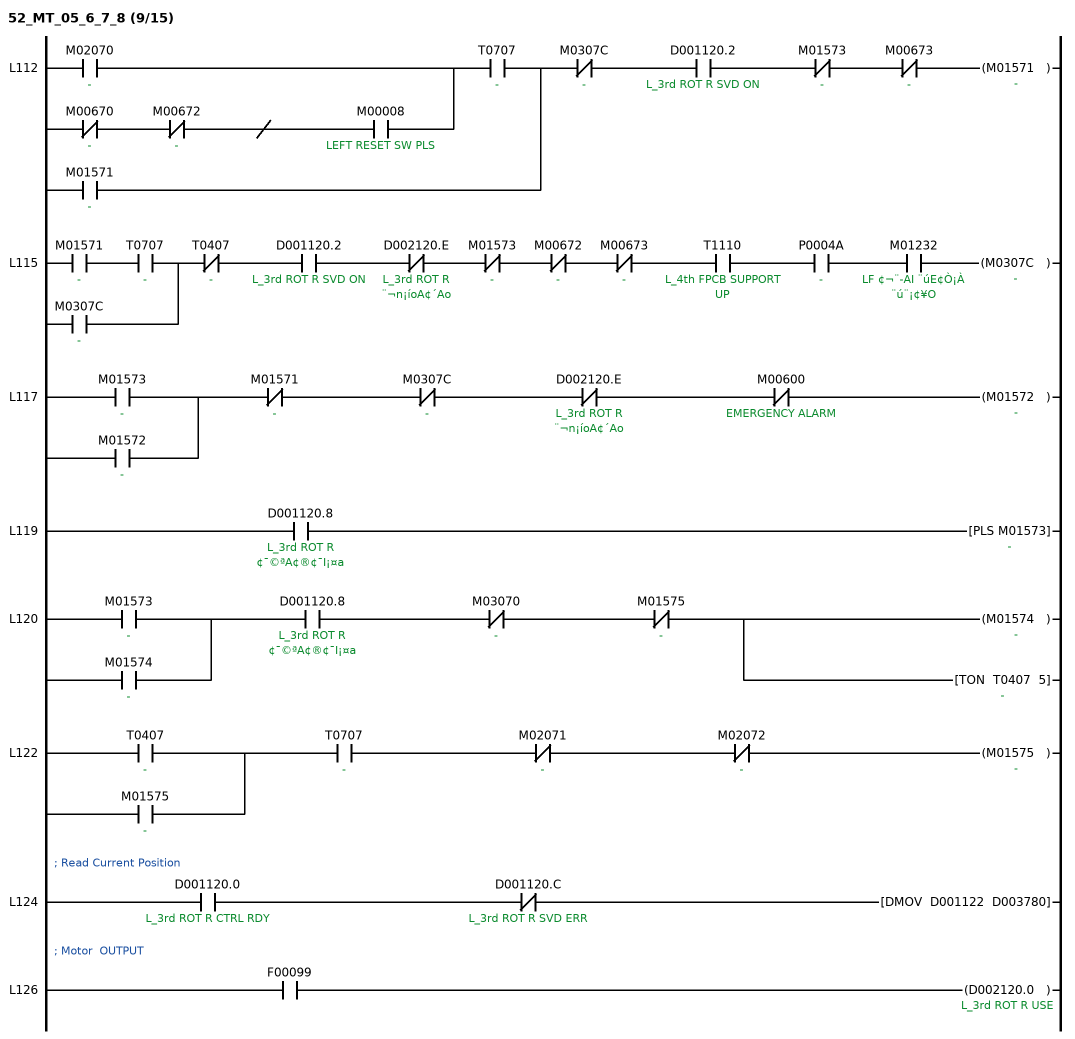
[picture p264: 52_MT_05_6_7_8 rungs L112-L126]
; L112
LOAD      M02070	// -
LOAD NOT  M00670	// -
AND NOT   M00672	// -
NOT
AND       M00008	// LEFT RESET SW PLS
OR LOAD
AND       T0707	// -
OR        M01571	// -
AND NOT   M0307C	// -
AND       D001120.2	// L_3rd ROT R SVD ON
AND NOT   M01573	// -
AND NOT   M00673	// -
OUT       M01571	// -
; L115
LOAD      M01571	// -
AND       T0707	// -
OR        M0307C	// -
AND NOT   T0407	// -
AND       D001120.2	// L_3rd ROT R SVD ON
AND NOT   D002120.E	// L_3rd ROT R ¨¬n¡íoA¢´Ao
AND NOT   M01573	// -
AND NOT   M00672	// -
AND NOT   M00673	// -
AND       T1110	// L_4th FPCB SUPPORT UP
AND       P0004A	// -
AND       M01232	// LF ¢¬¨­AI ¨úE¢Ò¡À ¨ú¨¡¢¥O
OUT       M0307C	// -
; L117
LOAD      M01573	// -
OR        M01572	// -
AND NOT   M01571	// -
AND NOT   M0307C	// -
AND NOT   D002120.E	// L_3rd ROT R ¨¬n¡íoA¢´Ao
AND NOT   M00600	// EMERGENCY ALARM
OUT       M01572	// -
; L119
LOAD      D001120.8	// L_3rd ROT R ¢¯©ªA¢®¢¯I¡¤a
OUTP      M01573	// -
; L120
LOAD      M01573	// -
OR        M01574	// -
AND       D001120.8	// L_3rd ROT R ¢¯©ªA¢®¢¯I¡¤a
AND NOT   M03070	// -
AND NOT   M01575	// -
OUT       M01574	// -
TON       T0407 5	// -
; L122
LOAD      T0407	// -
OR        M01575	// -
AND       T0707	// -
AND NOT   M02071	// -
AND NOT   M02072	// -
OUT       M01575	// -
; L124
LOAD      D001120.0	// L_3rd ROT R CTRL RDY
AND NOT   D001120.C	// L_3rd ROT R SVD ERR
DMOV      D001122 D003780
// output comment: Read Current Position
//  Motor  OUTPUT
; L126
LOAD      F00099
OUT       D002120.0	// L_3rd ROT R USE

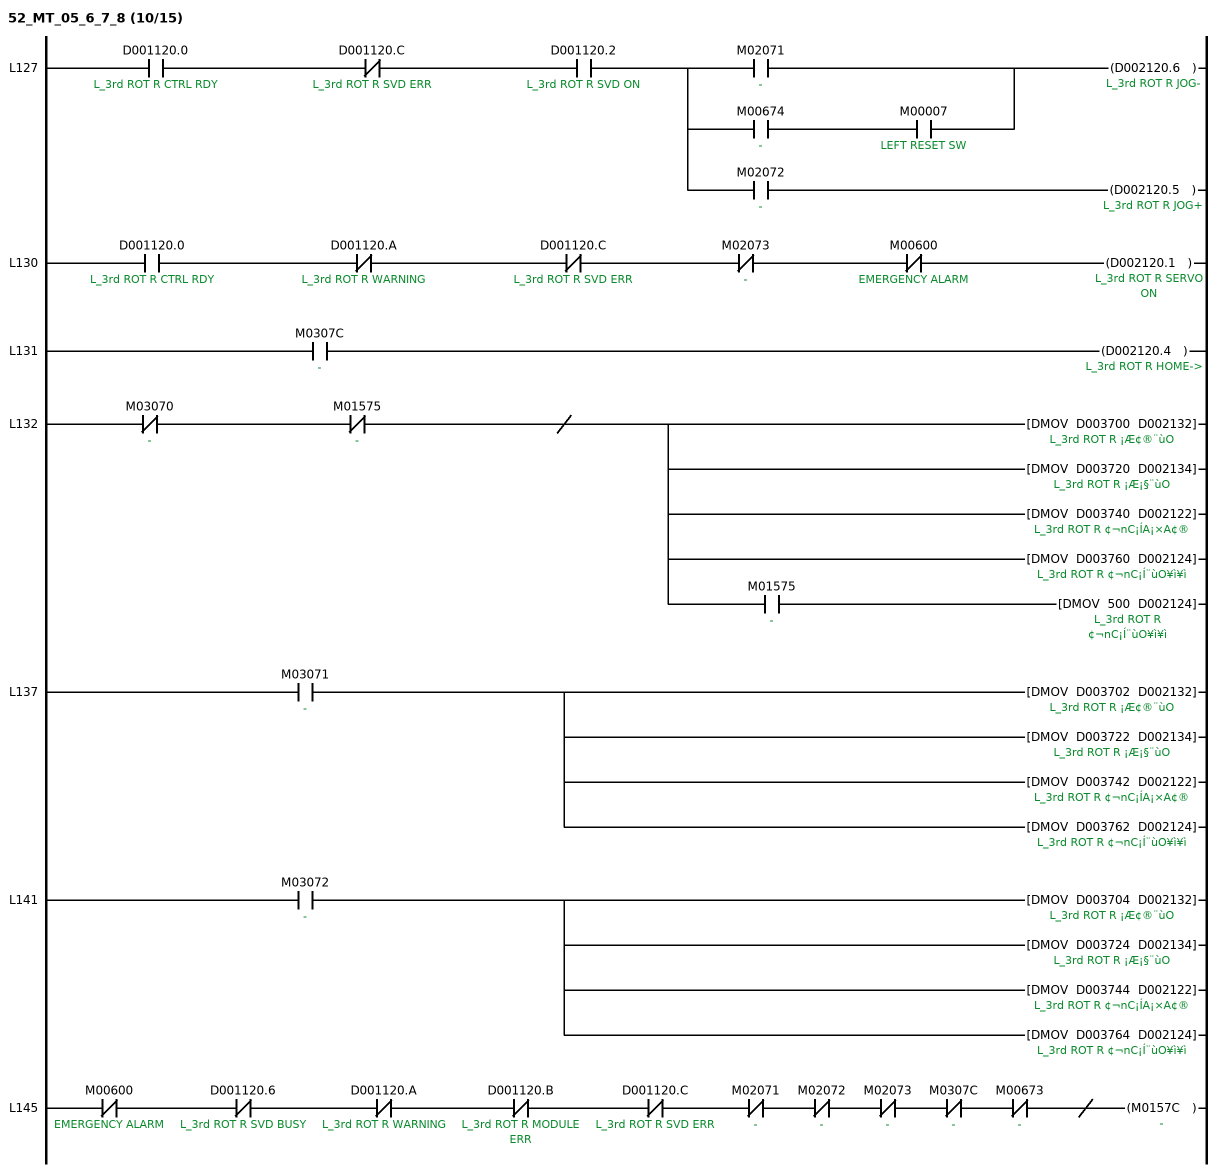
; L127
LOAD      D001120.0	// L_3rd ROT R CTRL RDY
AND NOT   D001120.C	// L_3rd ROT R SVD ERR
AND       D001120.2	// L_3rd ROT R SVD ON
MPUSH
LOAD      M02071	// -
LOAD      M00674	// -
AND       M00007	// LEFT RESET SW
OR LOAD
AND LOAD
OUT       D002120.6	// L_3rd ROT R JOG-
MPOP
AND       M02072	// -
OUT       D002120.5	// L_3rd ROT R JOG+
; L130
LOAD      D001120.0	// L_3rd ROT R CTRL RDY
AND NOT   D001120.A	// L_3rd ROT R WARNING
AND NOT   D001120.C	// L_3rd ROT R SVD ERR
AND NOT   M02073	// -
AND NOT   M00600	// EMERGENCY ALARM
OUT       D002120.1	// L_3rd ROT R SERVO ON
; L131
LOAD      M0307C	// -
OUT       D002120.4	// L_3rd ROT R HOME->
; L132
LOAD NOT  M03070	// -
AND NOT   M01575	// -
NOT
DMOV      D003700 D002132	// L_3rd ROT R ¡Æ¢®¨ùO
DMOV      D003720 D002134	// L_3rd ROT R ¡Æ¡§¨ùO
DMOV      D003740 D002122	// L_3rd ROT R ¢¬nC¡ÍA¡×A¢®
DMOV      D003760 D002124	// L_3rd ROT R ¢¬nC¡Í¨ùO¥ì¥ì
AND       M01575	// -
DMOV      500 D002124	// L_3rd ROT R ¢¬nC¡Í¨ùO¥ì¥ì
; L137
LOAD      M03071	// -
DMOV      D003702 D002132	// L_3rd ROT R ¡Æ¢®¨ùO
DMOV      D003722 D002134	// L_3rd ROT R ¡Æ¡§¨ùO
DMOV      D003742 D002122	// L_3rd ROT R ¢¬nC¡ÍA¡×A¢®
DMOV      D003762 D002124	// L_3rd ROT R ¢¬nC¡Í¨ùO¥ì¥ì
; L141
LOAD      M03072	// -
DMOV      D003704 D002132	// L_3rd ROT R ¡Æ¢®¨ùO
DMOV      D003724 D002134	// L_3rd ROT R ¡Æ¡§¨ùO
DMOV      D003744 D002122	// L_3rd ROT R ¢¬nC¡ÍA¡×A¢®
DMOV      D003764 D002124	// L_3rd ROT R ¢¬nC¡Í¨ùO¥ì¥ì
; L145
LOAD NOT  M00600	// EMERGENCY ALARM
AND NOT   D001120.6	// L_3rd ROT R SVD BUSY
AND NOT   D001120.A	// L_3rd ROT R WARNING
AND NOT   D001120.B	// L_3rd ROT R MODULE ERR
AND NOT   D001120.C	// L_3rd ROT R SVD ERR
AND NOT   M02071	// -
AND NOT   M02072	// -
AND NOT   M02073	// -
AND NOT   M0307C	// -
AND NOT   M00673	// -
NOT
OUT       M0157C	// -

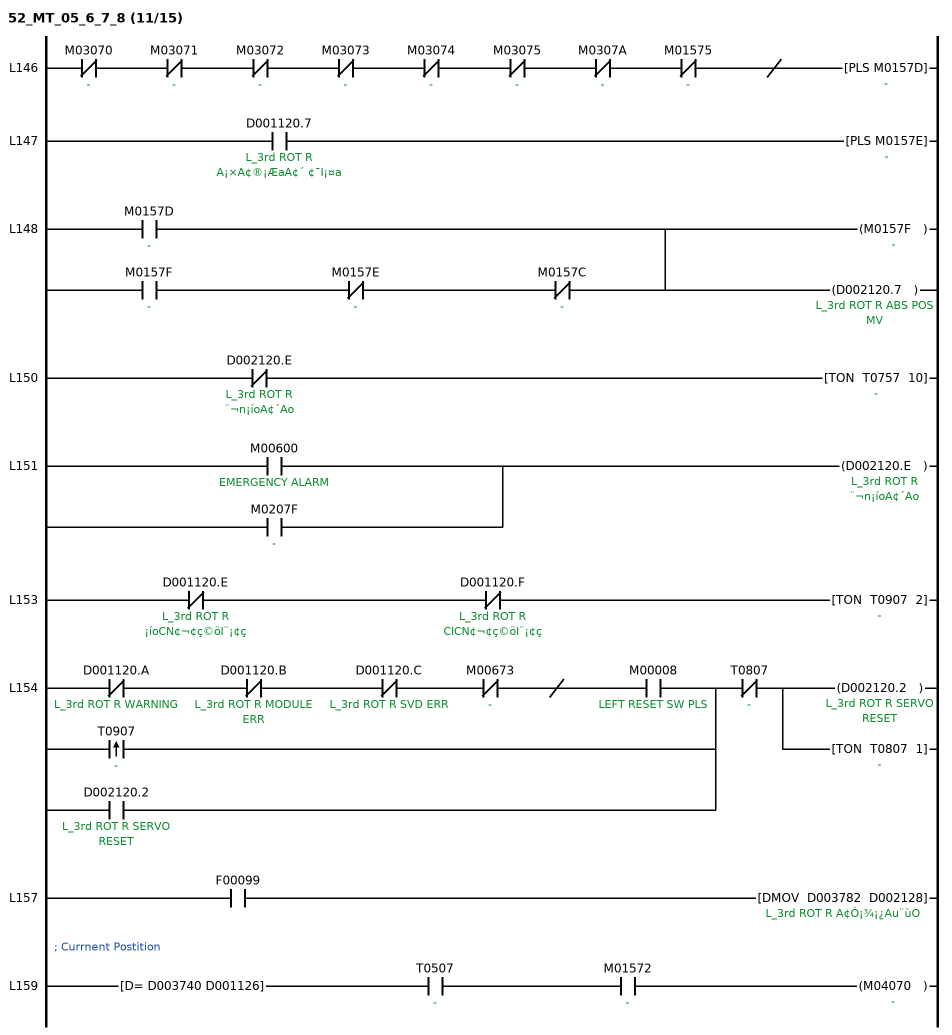
; L146
LOAD NOT  M03070	// -
AND NOT   M03071	// -
AND NOT   M03072	// -
AND NOT   M03073	// -
AND NOT   M03074	// -
AND NOT   M03075	// -
AND NOT   M0307A	// -
AND NOT   M01575	// -
NOT
OUTP      M0157D	// -
; L147
LOAD      D001120.7	// L_3rd ROT R A¡×A¢®¡ÆaA¢´ ¢¯I¡¤a
OUTP      M0157E	// -
; L148
LOAD      M0157D	// -
LOAD      M0157F	// -
AND NOT   M0157E	// -
AND NOT   M0157C	// -
OR LOAD
OUT       M0157F	// -
OUT       D002120.7	// L_3rd ROT R ABS POS MV
; L150
LOAD NOT  D002120.E	// L_3rd ROT R ¨¬n¡íoA¢´Ao
TON       T0757 10	// -
; L151
LOAD      M00600	// EMERGENCY ALARM
OR        M0207F	// -
OUT       D002120.E	// L_3rd ROT R ¨¬n¡íoA¢´Ao
; L153
LOAD NOT  D001120.E	// L_3rd ROT R ¡íoCN¢¬¢ç©öI¨¡¢ç
AND NOT   D001120.F	// L_3rd ROT R CICN¢¬¢ç©öI¨¡¢ç
TON       T0907 2	// -
; L154
LOAD NOT  D001120.A	// L_3rd ROT R WARNING
AND NOT   D001120.B	// L_3rd ROT R MODULE ERR
AND NOT   D001120.C	// L_3rd ROT R SVD ERR
AND NOT   M00673	// -
NOT
AND       M00008	// LEFT RESET SW PLS
ORP       T0907	// -
OR        D002120.2	// L_3rd ROT R SERVO RESET
AND NOT   T0807	// -
OUT       D002120.2	// L_3rd ROT R SERVO RESET
TON       T0807 1	// -
; L157
LOAD      F00099
DMOV      D003782 D002128	// L_3rd ROT R A¢Ò¡¾¡¿Au¨ùO
// Currnent Postition
; L159
LOADD=    D003740 D001126
AND       T0507	// -
AND       M01572	// -
OUT       M04070	// -

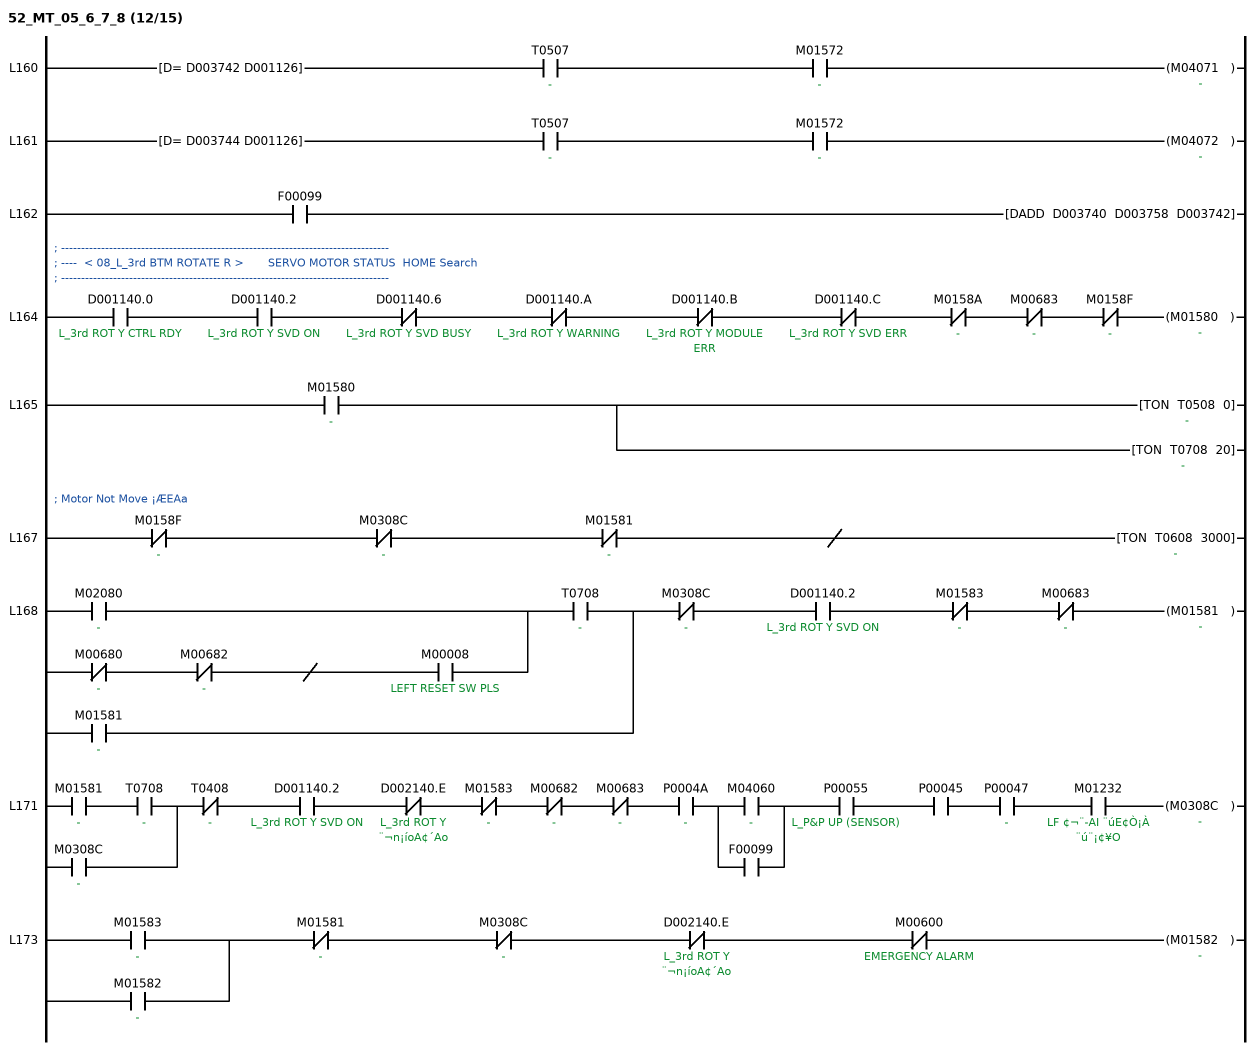
; L160
LOADD=    D003742 D001126
AND       T0507	// -
AND       M01572	// -
OUT       M04071	// -
; L161
LOADD=    D003744 D001126
AND       T0507	// -
AND       M01572	// -
OUT       M04072	// -
; L162
LOAD      F00099
DADD      D003740 D003758 D003742
// ----------------------------------------------------------------------------------
// 
// ----  < 08_L_3rd BTM ROTATE R >       SERVO MOTOR STATUS  HOME Search
// 
// ----------------------------------------------------------------------------------
; L164
LOAD      D001140.0	// L_3rd ROT Y CTRL RDY
AND       D001140.2	// L_3rd ROT Y SVD ON
AND NOT   D001140.6	// L_3rd ROT Y SVD BUSY
AND NOT   D001140.A	// L_3rd ROT Y WARNING
AND NOT   D001140.B	// L_3rd ROT Y MODULE ERR
AND NOT   D001140.C	// L_3rd ROT Y SVD ERR
AND NOT   M0158A	// -
AND NOT   M00683	// -
AND NOT   M0158F	// -
OUT       M01580	// -
; L165
LOAD      M01580	// -
TON       T0508 0	// -
TON       T0708 20	// -
; L167
LOAD NOT  M0158F	// -
AND NOT   M0308C	// -
AND NOT   M01581	// -
NOT
TON       T0608 3000	// -
// output comment: Motor Not Move ¡ÆEAa
; L168
LOAD      M02080	// -
LOAD NOT  M00680	// -
AND NOT   M00682	// -
NOT
AND       M00008	// LEFT RESET SW PLS
OR LOAD
AND       T0708	// -
OR        M01581	// -
AND NOT   M0308C	// -
AND       D001140.2	// L_3rd ROT Y SVD ON
AND NOT   M01583	// -
AND NOT   M00683	// -
OUT       M01581	// -
; L171
LOAD      M01581	// -
AND       T0708	// -
OR        M0308C	// -
AND NOT   T0408	// -
AND       D001140.2	// L_3rd ROT Y SVD ON
AND NOT   D002140.E	// L_3rd ROT Y ¨¬n¡íoA¢´Ao
AND NOT   M01583	// -
AND NOT   M00682	// -
AND NOT   M00683	// -
AND       P0004A	// -
LOAD      M04060	// -
OR        F00099
AND LOAD
AND       P00055	// L_P&P UP (SENSOR)
AND       P00045
AND       P00047	// -
AND       M01232	// LF ¢¬¨­AI ¨úE¢Ò¡À ¨ú¨¡¢¥O
OUT       M0308C	// -
; L173
LOAD      M01583	// -
OR        M01582	// -
AND NOT   M01581	// -
AND NOT   M0308C	// -
AND NOT   D002140.E	// L_3rd ROT Y ¨¬n¡íoA¢´Ao
AND NOT   M00600	// EMERGENCY ALARM
OUT       M01582	// -

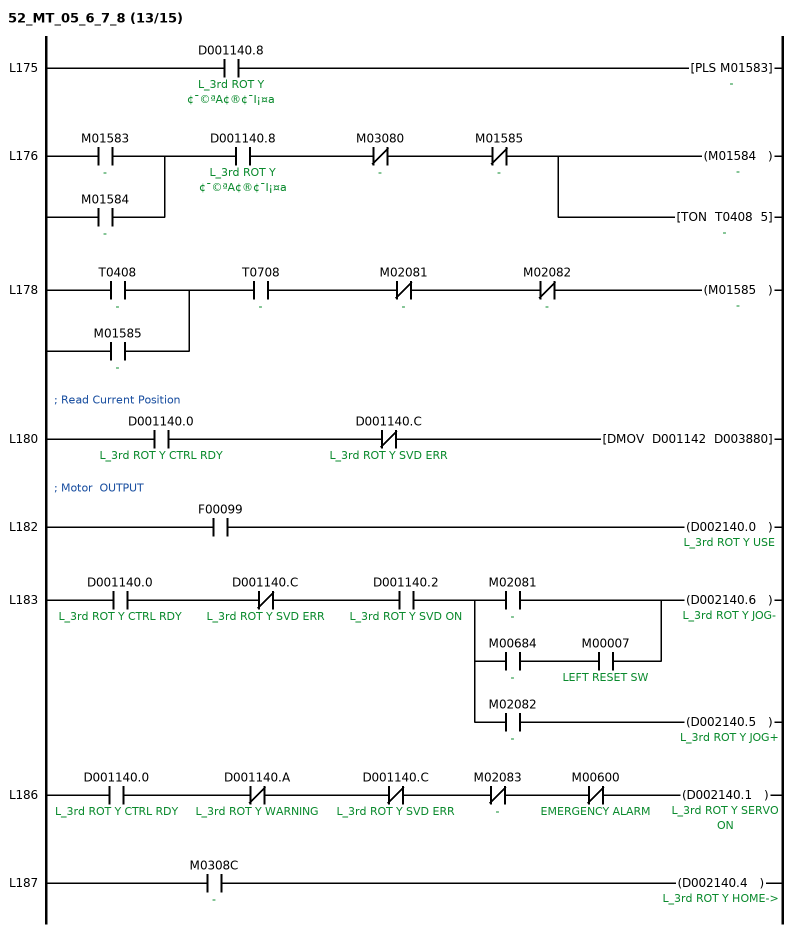
; L175
LOAD      D001140.8	// L_3rd ROT Y ¢¯©ªA¢®¢¯I¡¤a
OUTP      M01583	// -
; L176
LOAD      M01583	// -
OR        M01584	// -
AND       D001140.8	// L_3rd ROT Y ¢¯©ªA¢®¢¯I¡¤a
AND NOT   M03080	// -
AND NOT   M01585	// -
OUT       M01584	// -
TON       T0408 5	// -
; L178
LOAD      T0408	// -
OR        M01585	// -
AND       T0708	// -
AND NOT   M02081	// -
AND NOT   M02082	// -
OUT       M01585	// -
; L180
LOAD      D001140.0	// L_3rd ROT Y CTRL RDY
AND NOT   D001140.C	// L_3rd ROT Y SVD ERR
DMOV      D001142 D003880
// output comment: Read Current Position
//  Motor  OUTPUT
; L182
LOAD      F00099
OUT       D002140.0	// L_3rd ROT Y USE
; L183
LOAD      D001140.0	// L_3rd ROT Y CTRL RDY
AND NOT   D001140.C	// L_3rd ROT Y SVD ERR
AND       D001140.2	// L_3rd ROT Y SVD ON
MPUSH
LOAD      M02081	// -
LOAD      M00684	// -
AND       M00007	// LEFT RESET SW
OR LOAD
AND LOAD
OUT       D002140.6	// L_3rd ROT Y JOG-
MPOP
AND       M02082	// -
OUT       D002140.5	// L_3rd ROT Y JOG+
; L186
LOAD      D001140.0	// L_3rd ROT Y CTRL RDY
AND NOT   D001140.A	// L_3rd ROT Y WARNING
AND NOT   D001140.C	// L_3rd ROT Y SVD ERR
AND NOT   M02083	// -
AND NOT   M00600	// EMERGENCY ALARM
OUT       D002140.1	// L_3rd ROT Y SERVO ON
; L187
LOAD      M0308C	// -
OUT       D002140.4	// L_3rd ROT Y HOME->

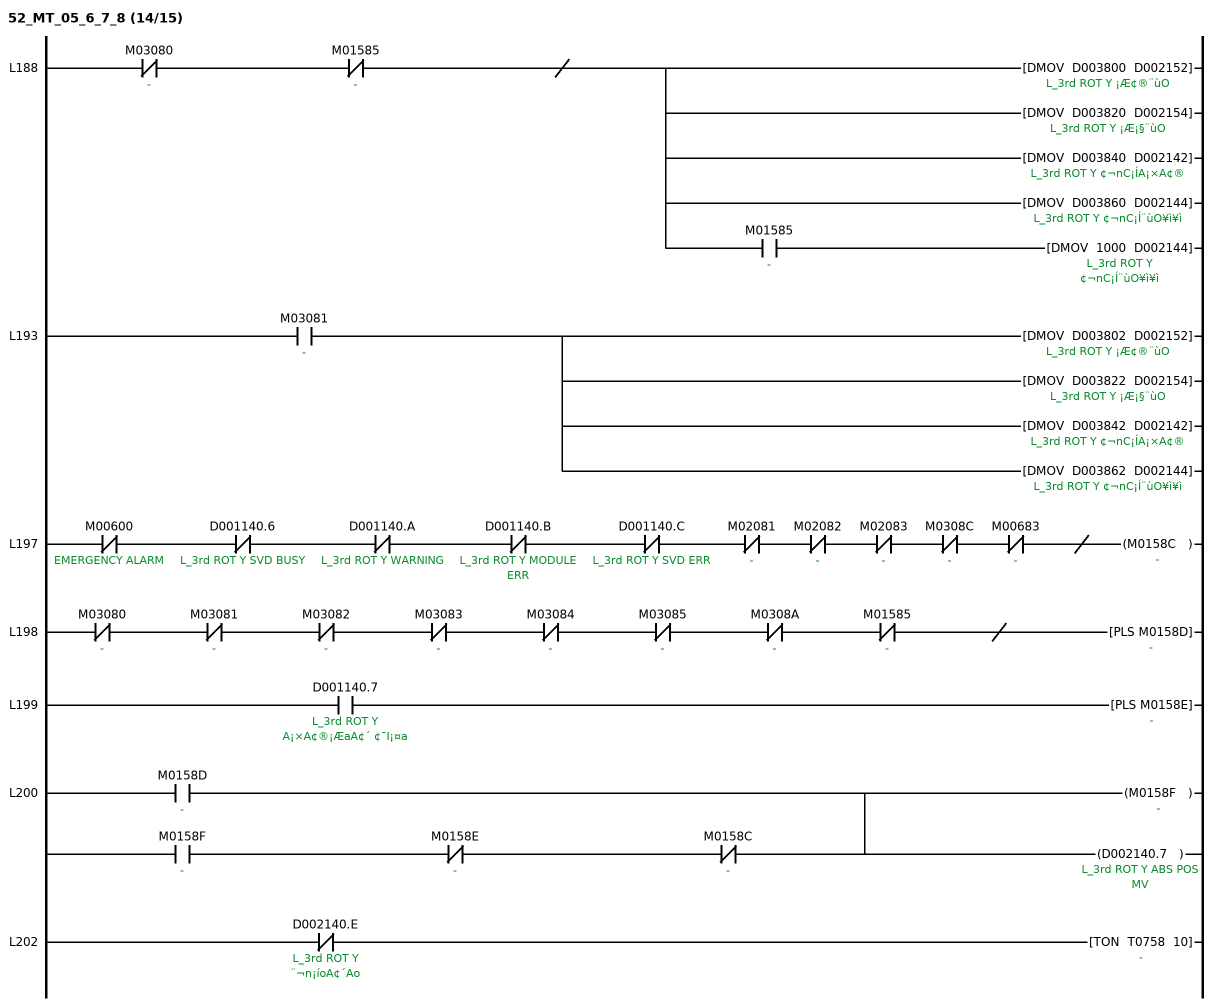
; L188
LOAD NOT  M03080	// -
AND NOT   M01585	// -
NOT
DMOV      D003800 D002152	// L_3rd ROT Y ¡Æ¢®¨ùO
DMOV      D003820 D002154	// L_3rd ROT Y ¡Æ¡§¨ùO
DMOV      D003840 D002142	// L_3rd ROT Y ¢¬nC¡ÍA¡×A¢®
DMOV      D003860 D002144	// L_3rd ROT Y ¢¬nC¡Í¨ùO¥ì¥ì
AND       M01585	// -
DMOV      1000 D002144	// L_3rd ROT Y ¢¬nC¡Í¨ùO¥ì¥ì
; L193
LOAD      M03081	// -
DMOV      D003802 D002152	// L_3rd ROT Y ¡Æ¢®¨ùO
DMOV      D003822 D002154	// L_3rd ROT Y ¡Æ¡§¨ùO
DMOV      D003842 D002142	// L_3rd ROT Y ¢¬nC¡ÍA¡×A¢®
DMOV      D003862 D002144	// L_3rd ROT Y ¢¬nC¡Í¨ùO¥ì¥ì
; L197
LOAD NOT  M00600	// EMERGENCY ALARM
AND NOT   D001140.6	// L_3rd ROT Y SVD BUSY
AND NOT   D001140.A	// L_3rd ROT Y WARNING
AND NOT   D001140.B	// L_3rd ROT Y MODULE ERR
AND NOT   D001140.C	// L_3rd ROT Y SVD ERR
AND NOT   M02081	// -
AND NOT   M02082	// -
AND NOT   M02083	// -
AND NOT   M0308C	// -
AND NOT   M00683	// -
NOT
OUT       M0158C	// -
; L198
LOAD NOT  M03080	// -
AND NOT   M03081	// -
AND NOT   M03082	// -
AND NOT   M03083	// -
AND NOT   M03084	// -
AND NOT   M03085	// -
AND NOT   M0308A	// -
AND NOT   M01585	// -
NOT
OUTP      M0158D	// -
; L199
LOAD      D001140.7	// L_3rd ROT Y A¡×A¢®¡ÆaA¢´ ¢¯I¡¤a
OUTP      M0158E	// -
; L200
LOAD      M0158D	// -
LOAD      M0158F	// -
AND NOT   M0158E	// -
AND NOT   M0158C	// -
OR LOAD
OUT       M0158F	// -
OUT       D002140.7	// L_3rd ROT Y ABS POS MV
; L202
LOAD NOT  D002140.E	// L_3rd ROT Y ¨¬n¡íoA¢´Ao
TON       T0758 10	// -

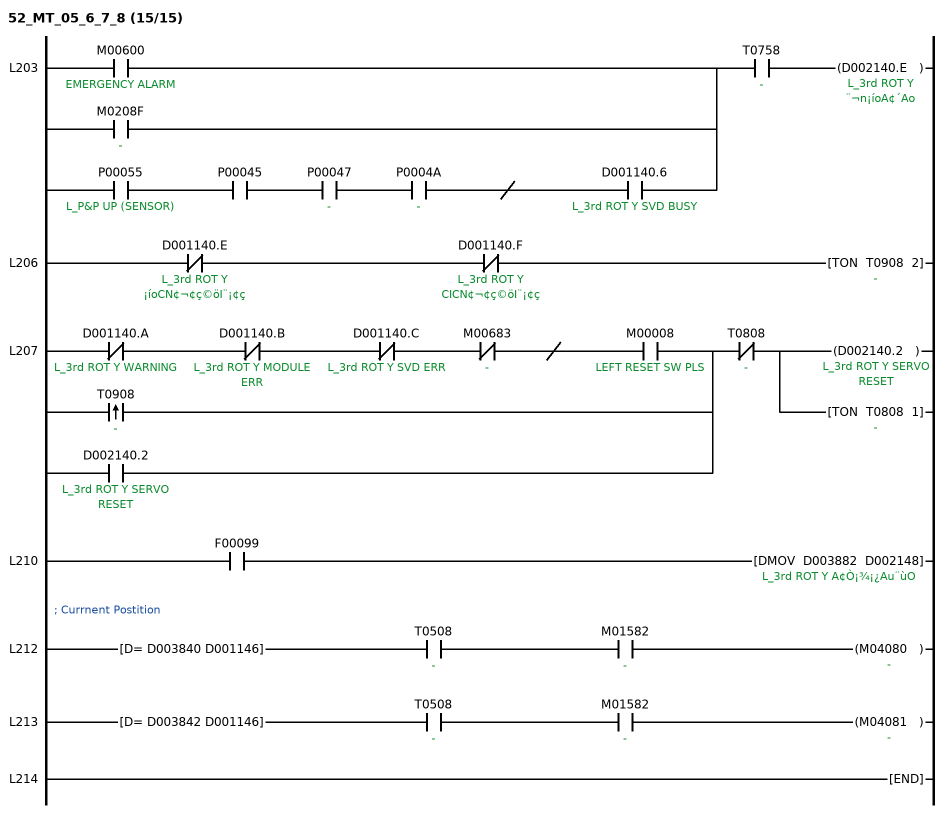
; L203
LOAD      M00600	// EMERGENCY ALARM
OR        M0208F	// -
LOAD      P00055	// L_P&P UP (SENSOR)
AND       P00045
AND       P00047	// -
AND       P0004A	// -
NOT
AND       D001140.6	// L_3rd ROT Y SVD BUSY
OR LOAD
AND       T0758	// -
OUT       D002140.E	// L_3rd ROT Y ¨¬n¡íoA¢´Ao
; L206
LOAD NOT  D001140.E	// L_3rd ROT Y ¡íoCN¢¬¢ç©öI¨¡¢ç
AND NOT   D001140.F	// L_3rd ROT Y CICN¢¬¢ç©öI¨¡¢ç
TON       T0908 2	// -
; L207
LOAD NOT  D001140.A	// L_3rd ROT Y WARNING
AND NOT   D001140.B	// L_3rd ROT Y MODULE ERR
AND NOT   D001140.C	// L_3rd ROT Y SVD ERR
AND NOT   M00683	// -
NOT
AND       M00008	// LEFT RESET SW PLS
ORP       T0908	// -
OR        D002140.2	// L_3rd ROT Y SERVO RESET
AND NOT   T0808	// -
OUT       D002140.2	// L_3rd ROT Y SERVO RESET
TON       T0808 1	// -
; L210
LOAD      F00099
DMOV      D003882 D002148	// L_3rd ROT Y A¢Ò¡¾¡¿Au¨ùO
// Currnent Postition
; L212
LOADD=    D003840 D001146
AND       T0508	// -
AND       M01582	// -
OUT       M04080	// -
; L213
LOADD=    D003842 D001146
AND       T0508	// -
AND       M01582	// -
OUT       M04081	// -
; L214
END

PROGRAM 53_MT_09_10_11_12 (task: ¨ö¨¬A¥ì CA¡¤I¡¾¡¿¡¤¡Í)

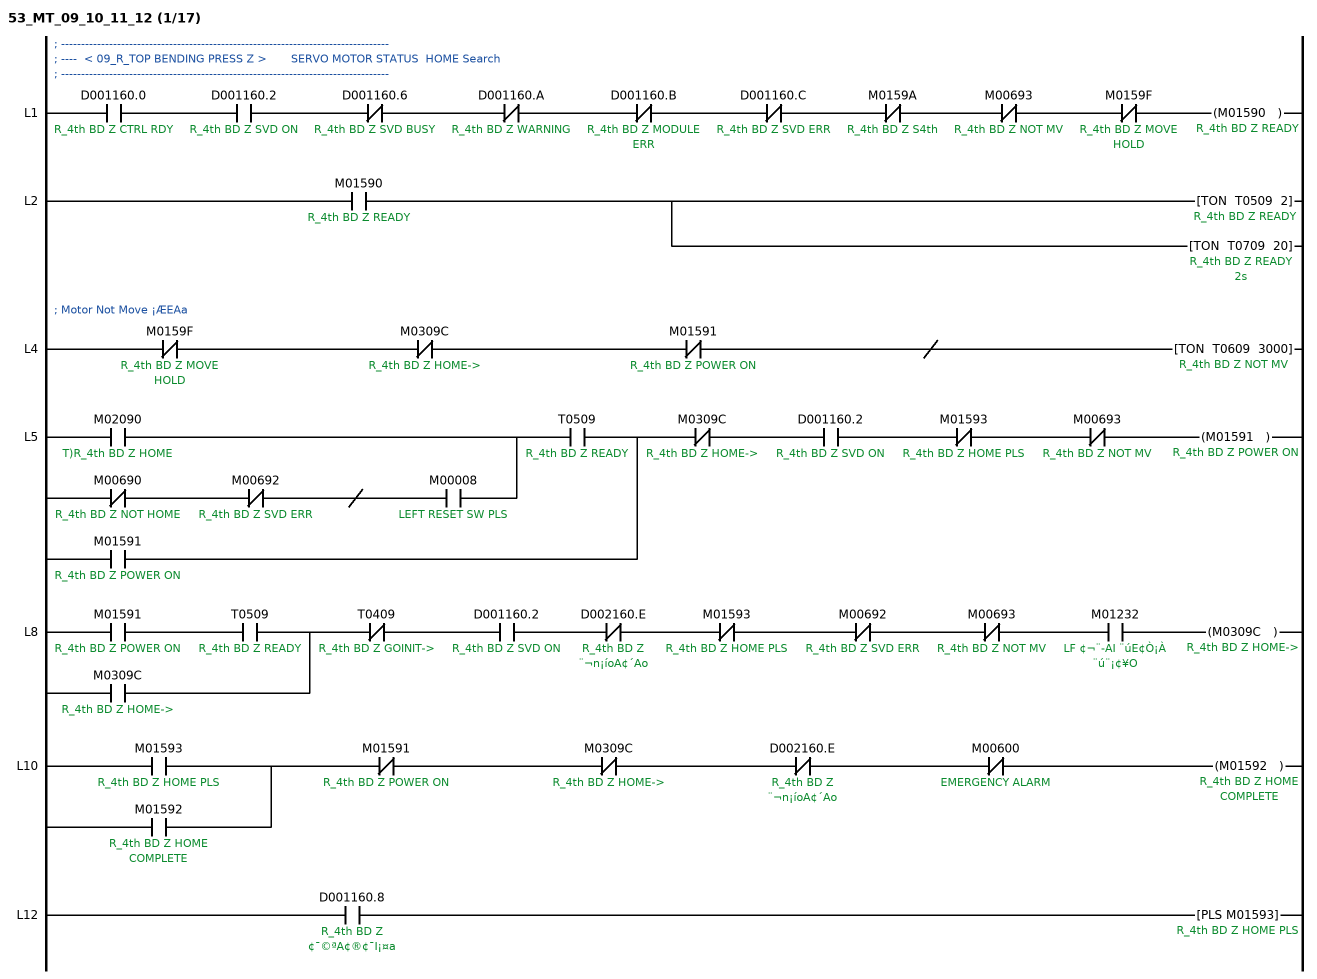
// ----------------------------------------------------------------------------------
// 
// ----  < 09_R_TOP BENDING PRESS Z >       SERVO MOTOR STATUS  HOME Search
// 
// ----------------------------------------------------------------------------------
; L1
LOAD      D001160.0	// R_4th BD Z CTRL RDY
AND       D001160.2	// R_4th BD Z SVD ON
AND NOT   D001160.6	// R_4th BD Z SVD BUSY
AND NOT   D001160.A	// R_4th BD Z WARNING
AND NOT   D001160.B	// R_4th BD Z MODULE ERR
AND NOT   D001160.C	// R_4th BD Z SVD ERR
AND NOT   M0159A	// R_4th BD Z S4th
AND NOT   M00693	// R_4th BD Z NOT MV
AND NOT   M0159F	// R_4th BD Z MOVE HOLD
OUT       M01590	// R_4th BD Z READY
; L2
LOAD      M01590	// R_4th BD Z READY
TON       T0509 2	// R_4th BD Z READY
TON       T0709 20	// R_4th BD Z READY 2s
; L4
LOAD NOT  M0159F	// R_4th BD Z MOVE HOLD
AND NOT   M0309C	// R_4th BD Z HOME->
AND NOT   M01591	// R_4th BD Z POWER ON
NOT
TON       T0609 3000	// R_4th BD Z NOT MV
// output comment: Motor Not Move ¡ÆEAa
; L5
LOAD      M02090	// T)R_4th BD Z HOME
LOAD NOT  M00690	// R_4th BD Z NOT HOME
AND NOT   M00692	// R_4th BD Z SVD ERR
NOT
AND       M00008	// LEFT RESET SW PLS
OR LOAD
AND       T0509	// R_4th BD Z READY
OR        M01591	// R_4th BD Z POWER ON
AND NOT   M0309C	// R_4th BD Z HOME->
AND       D001160.2	// R_4th BD Z SVD ON
AND NOT   M01593	// R_4th BD Z HOME PLS
AND NOT   M00693	// R_4th BD Z NOT MV
OUT       M01591	// R_4th BD Z POWER ON
; L8
LOAD      M01591	// R_4th BD Z POWER ON
AND       T0509	// R_4th BD Z READY
OR        M0309C	// R_4th BD Z HOME->
AND NOT   T0409	// R_4th BD Z GOINIT->
AND       D001160.2	// R_4th BD Z SVD ON
AND NOT   D002160.E	// R_4th BD Z ¨¬n¡íoA¢´Ao
AND NOT   M01593	// R_4th BD Z HOME PLS
AND NOT   M00692	// R_4th BD Z SVD ERR
AND NOT   M00693	// R_4th BD Z NOT MV
AND       M01232	// LF ¢¬¨­AI ¨úE¢Ò¡À ¨ú¨¡¢¥O
OUT       M0309C	// R_4th BD Z HOME->
; L10
LOAD      M01593	// R_4th BD Z HOME PLS
OR        M01592	// R_4th BD Z HOME COMPLETE
AND NOT   M01591	// R_4th BD Z POWER ON
AND NOT   M0309C	// R_4th BD Z HOME->
AND NOT   D002160.E	// R_4th BD Z ¨¬n¡íoA¢´Ao
AND NOT   M00600	// EMERGENCY ALARM
OUT       M01592	// R_4th BD Z HOME COMPLETE
; L12
LOAD      D001160.8	// R_4th BD Z ¢¯©ªA¢®¢¯I¡¤a
OUTP      M01593	// R_4th BD Z HOME PLS

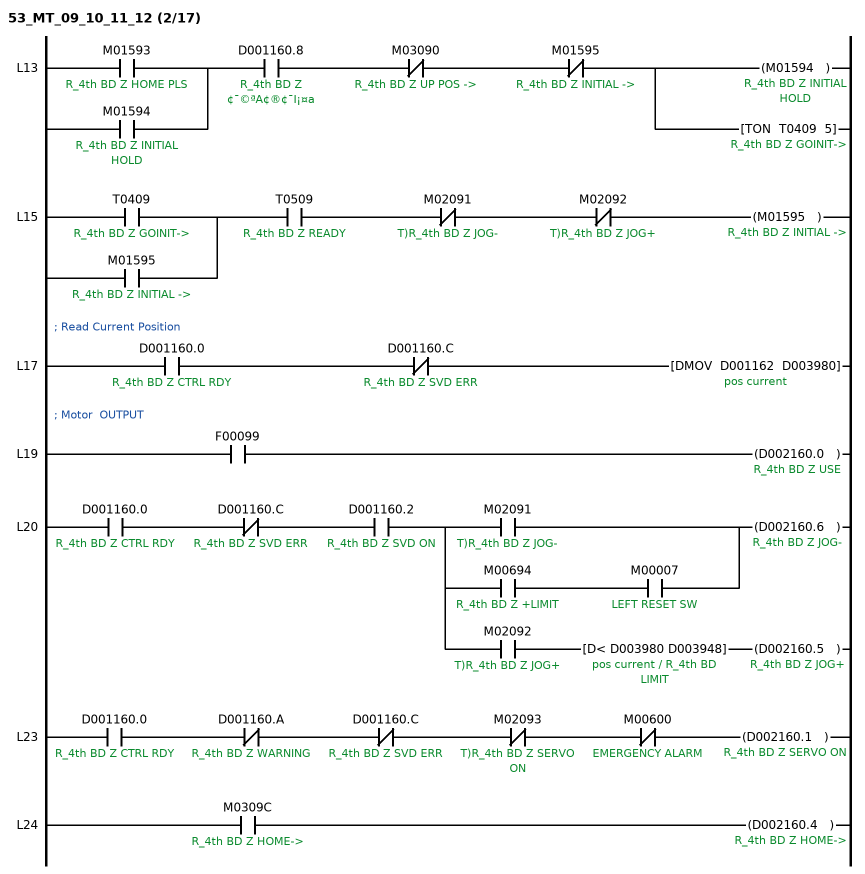
; L13
LOAD      M01593	// R_4th BD Z HOME PLS
OR        M01594	// R_4th BD Z INITIAL HOLD
AND       D001160.8	// R_4th BD Z ¢¯©ªA¢®¢¯I¡¤a
AND NOT   M03090	// R_4th BD Z UP POS ->
AND NOT   M01595	// R_4th BD Z INITIAL ->
OUT       M01594	// R_4th BD Z INITIAL HOLD
TON       T0409 5	// R_4th BD Z GOINIT->
; L15
LOAD      T0409	// R_4th BD Z GOINIT->
OR        M01595	// R_4th BD Z INITIAL ->
AND       T0509	// R_4th BD Z READY
AND NOT   M02091	// T)R_4th BD Z JOG-
AND NOT   M02092	// T)R_4th BD Z JOG+
OUT       M01595	// R_4th BD Z INITIAL ->
; L17
LOAD      D001160.0	// R_4th BD Z CTRL RDY
AND NOT   D001160.C	// R_4th BD Z SVD ERR
DMOV      D001162 D003980	// pos current
// output comment: Read Current Position
//  Motor  OUTPUT
; L19
LOAD      F00099
OUT       D002160.0	// R_4th BD Z USE
; L20
LOAD      D001160.0	// R_4th BD Z CTRL RDY
AND NOT   D001160.C	// R_4th BD Z SVD ERR
AND       D001160.2	// R_4th BD Z SVD ON
MPUSH
LOAD      M02091	// T)R_4th BD Z JOG-
LOAD      M00694	// R_4th BD Z +LIMIT
AND       M00007	// LEFT RESET SW
OR LOAD
AND LOAD
OUT       D002160.6	// R_4th BD Z JOG-
MPOP
AND       M02092	// T)R_4th BD Z JOG+
ANDD<     D003980 D003948	// pos current / R_4th BD LIMIT
OUT       D002160.5	// R_4th BD Z JOG+
; L23
LOAD      D001160.0	// R_4th BD Z CTRL RDY
AND NOT   D001160.A	// R_4th BD Z WARNING
AND NOT   D001160.C	// R_4th BD Z SVD ERR
AND NOT   M02093	// T)R_4th BD Z SERVO ON
AND NOT   M00600	// EMERGENCY ALARM
OUT       D002160.1	// R_4th BD Z SERVO ON
; L24
LOAD      M0309C	// R_4th BD Z HOME->
OUT       D002160.4	// R_4th BD Z HOME->

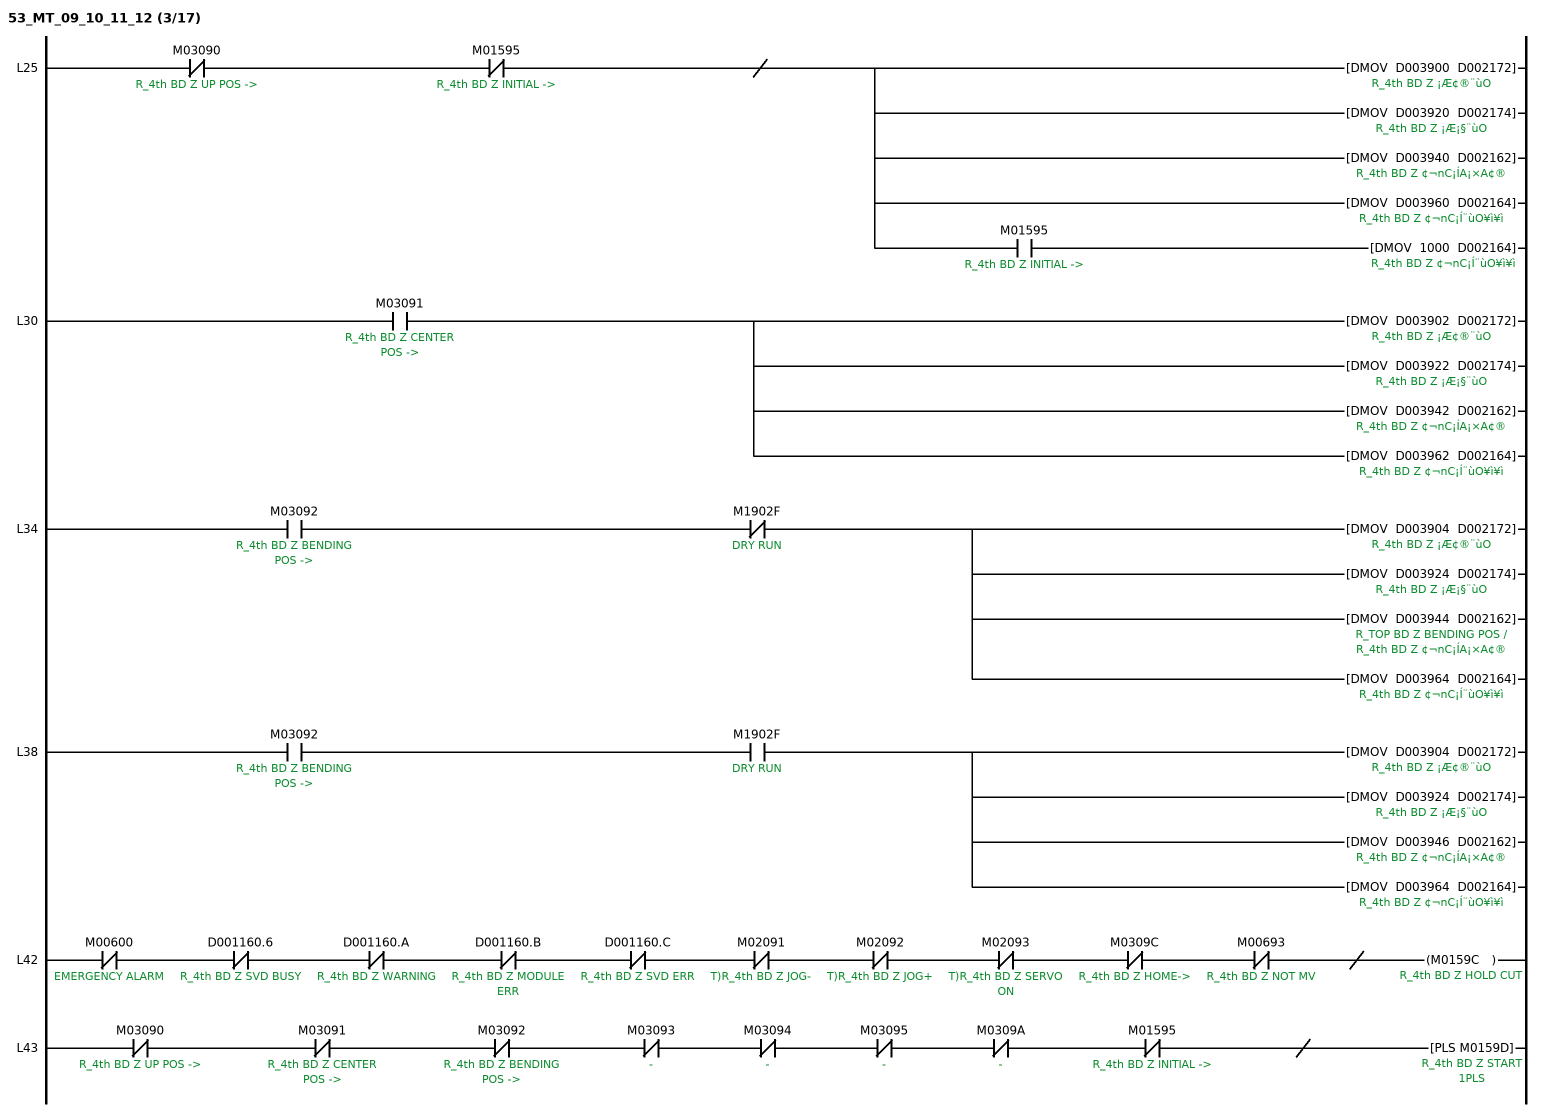
; L25
LOAD NOT  M03090	// R_4th BD Z UP POS ->
AND NOT   M01595	// R_4th BD Z INITIAL ->
NOT
DMOV      D003900 D002172	// R_4th BD Z ¡Æ¢®¨ùO
DMOV      D003920 D002174	// R_4th BD Z ¡Æ¡§¨ùO
DMOV      D003940 D002162	// R_4th BD Z ¢¬nC¡ÍA¡×A¢®
DMOV      D003960 D002164	// R_4th BD Z ¢¬nC¡Í¨ùO¥ì¥ì
AND       M01595	// R_4th BD Z INITIAL ->
DMOV      1000 D002164	// R_4th BD Z ¢¬nC¡Í¨ùO¥ì¥ì
; L30
LOAD      M03091	// R_4th BD Z CENTER POS ->
DMOV      D003902 D002172	// R_4th BD Z ¡Æ¢®¨ùO
DMOV      D003922 D002174	// R_4th BD Z ¡Æ¡§¨ùO
DMOV      D003942 D002162	// R_4th BD Z ¢¬nC¡ÍA¡×A¢®
DMOV      D003962 D002164	// R_4th BD Z ¢¬nC¡Í¨ùO¥ì¥ì
; L34
LOAD      M03092	// R_4th BD Z BENDING POS ->
AND NOT   M1902F	// DRY RUN
DMOV      D003904 D002172	// R_4th BD Z ¡Æ¢®¨ùO
DMOV      D003924 D002174	// R_4th BD Z ¡Æ¡§¨ùO
DMOV      D003944 D002162	// R_TOP BD Z BENDING POS / R_4th BD Z ¢¬nC¡ÍA¡×A¢®
DMOV      D003964 D002164	// R_4th BD Z ¢¬nC¡Í¨ùO¥ì¥ì
; L38
LOAD      M03092	// R_4th BD Z BENDING POS ->
AND       M1902F	// DRY RUN
DMOV      D003904 D002172	// R_4th BD Z ¡Æ¢®¨ùO
DMOV      D003924 D002174	// R_4th BD Z ¡Æ¡§¨ùO
DMOV      D003946 D002162	// R_4th BD Z ¢¬nC¡ÍA¡×A¢®
DMOV      D003964 D002164	// R_4th BD Z ¢¬nC¡Í¨ùO¥ì¥ì
; L42
LOAD NOT  M00600	// EMERGENCY ALARM
AND NOT   D001160.6	// R_4th BD Z SVD BUSY
AND NOT   D001160.A	// R_4th BD Z WARNING
AND NOT   D001160.B	// R_4th BD Z MODULE ERR
AND NOT   D001160.C	// R_4th BD Z SVD ERR
AND NOT   M02091	// T)R_4th BD Z JOG-
AND NOT   M02092	// T)R_4th BD Z JOG+
AND NOT   M02093	// T)R_4th BD Z SERVO ON
AND NOT   M0309C	// R_4th BD Z HOME->
AND NOT   M00693	// R_4th BD Z NOT MV
NOT
OUT       M0159C	// R_4th BD Z HOLD CUT
; L43
LOAD NOT  M03090	// R_4th BD Z UP POS ->
AND NOT   M03091	// R_4th BD Z CENTER POS ->
AND NOT   M03092	// R_4th BD Z BENDING POS ->
AND NOT   M03093	// -
AND NOT   M03094	// -
AND NOT   M03095	// -
AND NOT   M0309A	// -
AND NOT   M01595	// R_4th BD Z INITIAL ->
NOT
OUTP      M0159D	// R_4th BD Z START 1PLS

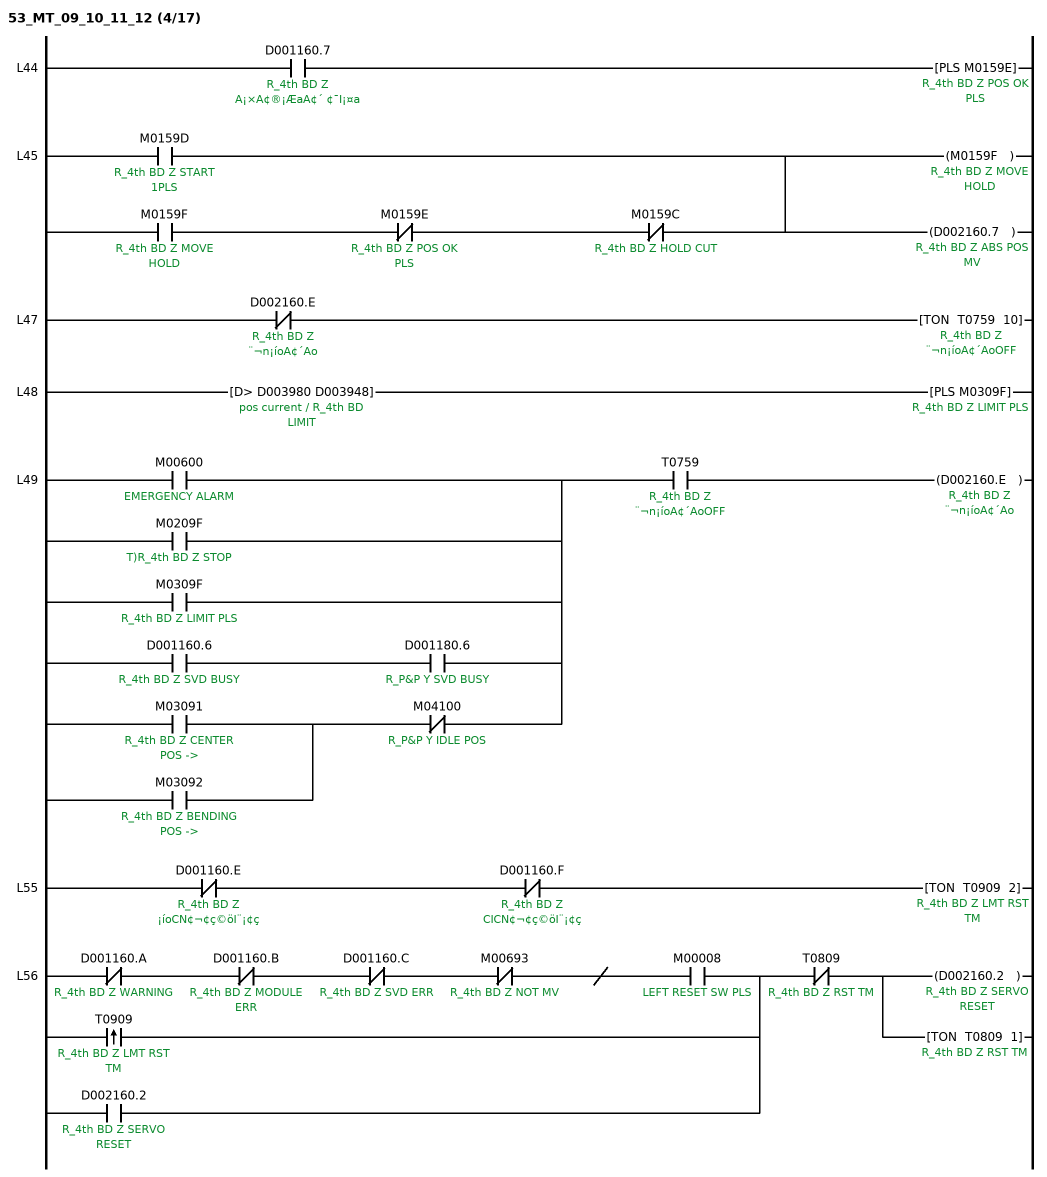
; L44
LOAD      D001160.7	// R_4th BD Z A¡×A¢®¡ÆaA¢´ ¢¯I¡¤a
OUTP      M0159E	// R_4th BD Z POS OK PLS
; L45
LOAD      M0159D	// R_4th BD Z START 1PLS
LOAD      M0159F	// R_4th BD Z MOVE HOLD
AND NOT   M0159E	// R_4th BD Z POS OK PLS
AND NOT   M0159C	// R_4th BD Z HOLD CUT
OR LOAD
OUT       M0159F	// R_4th BD Z MOVE HOLD
OUT       D002160.7	// R_4th BD Z ABS POS MV
; L47
LOAD NOT  D002160.E	// R_4th BD Z ¨¬n¡íoA¢´Ao
TON       T0759 10	// R_4th BD Z ¨¬n¡íoA¢´AoOFF
; L48
LOADD>    D003980 D003948	// pos current / R_4th BD LIMIT
OUTP      M0309F	// R_4th BD Z LIMIT PLS
; L49
LOAD      M00600	// EMERGENCY ALARM
OR        M0209F	// T)R_4th BD Z STOP
OR        M0309F	// R_4th BD Z LIMIT PLS
LOAD      D001160.6	// R_4th BD Z SVD BUSY
AND       D001180.6	// R_P&P Y SVD BUSY
OR LOAD
LOAD      M03091	// R_4th BD Z CENTER POS ->
OR        M03092	// R_4th BD Z BENDING POS ->
AND NOT   M04100	// R_P&P Y IDLE POS
OR LOAD
AND       T0759	// R_4th BD Z ¨¬n¡íoA¢´AoOFF
OUT       D002160.E	// R_4th BD Z ¨¬n¡íoA¢´Ao
; L55
LOAD NOT  D001160.E	// R_4th BD Z ¡íoCN¢¬¢ç©öI¨¡¢ç
AND NOT   D001160.F	// R_4th BD Z CICN¢¬¢ç©öI¨¡¢ç
TON       T0909 2	// R_4th BD Z LMT RST TM
; L56
LOAD NOT  D001160.A	// R_4th BD Z WARNING
AND NOT   D001160.B	// R_4th BD Z MODULE ERR
AND NOT   D001160.C	// R_4th BD Z SVD ERR
AND NOT   M00693	// R_4th BD Z NOT MV
NOT
AND       M00008	// LEFT RESET SW PLS
ORP       T0909	// R_4th BD Z LMT RST TM
OR        D002160.2	// R_4th BD Z SERVO RESET
AND NOT   T0809	// R_4th BD Z RST TM
OUT       D002160.2	// R_4th BD Z SERVO RESET
TON       T0809 1	// R_4th BD Z RST TM

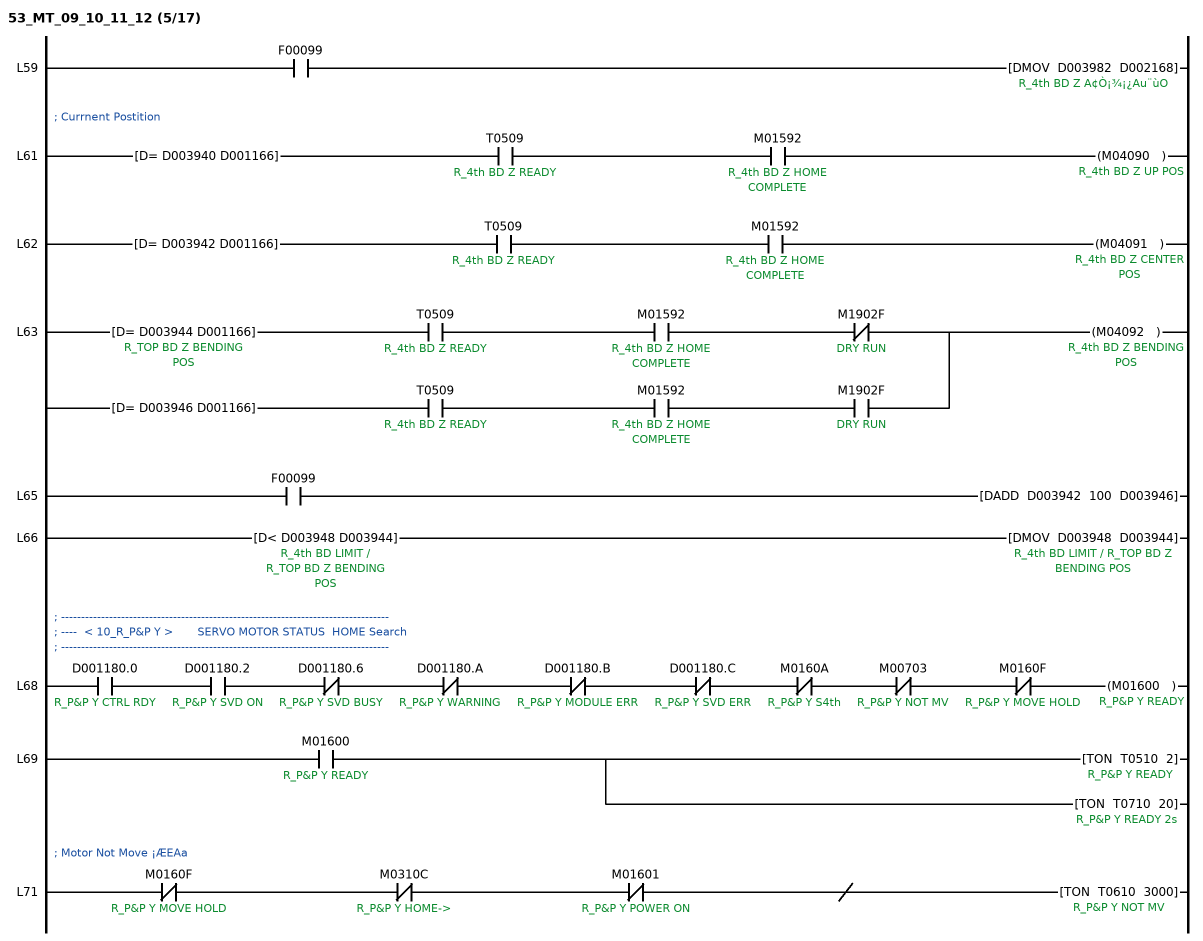
; L59
LOAD      F00099
DMOV      D003982 D002168	// R_4th BD Z A¢Ò¡¾¡¿Au¨ùO
// Currnent Postition
; L61
LOADD=    D003940 D001166
AND       T0509	// R_4th BD Z READY
AND       M01592	// R_4th BD Z HOME COMPLETE
OUT       M04090	// R_4th BD Z UP POS
; L62
LOADD=    D003942 D001166
AND       T0509	// R_4th BD Z READY
AND       M01592	// R_4th BD Z HOME COMPLETE
OUT       M04091	// R_4th BD Z CENTER POS
; L63
LOADD=    D003944 D001166	// R_TOP BD Z BENDING POS
AND       T0509	// R_4th BD Z READY
AND       M01592	// R_4th BD Z HOME COMPLETE
AND NOT   M1902F	// DRY RUN
LOADD=    D003946 D001166
AND       T0509	// R_4th BD Z READY
AND       M01592	// R_4th BD Z HOME COMPLETE
AND       M1902F	// DRY RUN
OR LOAD
OUT       M04092	// R_4th BD Z BENDING POS
; L65
LOAD      F00099
DADD      D003942 100 D003946
; L66
LOADD<    D003948 D003944	// R_4th BD LIMIT / R_TOP BD Z BENDING POS
DMOV      D003948 D003944	// R_4th BD LIMIT / R_TOP BD Z BENDING POS
// ----------------------------------------------------------------------------------
// 
// ----  < 10_R_P&P Y >       SERVO MOTOR STATUS  HOME Search
// 
// ----------------------------------------------------------------------------------
; L68
LOAD      D001180.0	// R_P&P Y CTRL RDY
AND       D001180.2	// R_P&P Y SVD ON
AND NOT   D001180.6	// R_P&P Y SVD BUSY
AND NOT   D001180.A	// R_P&P Y WARNING
AND NOT   D001180.B	// R_P&P Y MODULE ERR
AND NOT   D001180.C	// R_P&P Y SVD ERR
AND NOT   M0160A	// R_P&P Y S4th
AND NOT   M00703	// R_P&P Y NOT MV
AND NOT   M0160F	// R_P&P Y MOVE HOLD
OUT       M01600	// R_P&P Y READY
; L69
LOAD      M01600	// R_P&P Y READY
TON       T0510 2	// R_P&P Y READY
TON       T0710 20	// R_P&P Y READY 2s
; L71
LOAD NOT  M0160F	// R_P&P Y MOVE HOLD
AND NOT   M0310C	// R_P&P Y HOME->
AND NOT   M01601	// R_P&P Y POWER ON
NOT
TON       T0610 3000	// R_P&P Y NOT MV
// output comment: Motor Not Move ¡ÆEAa

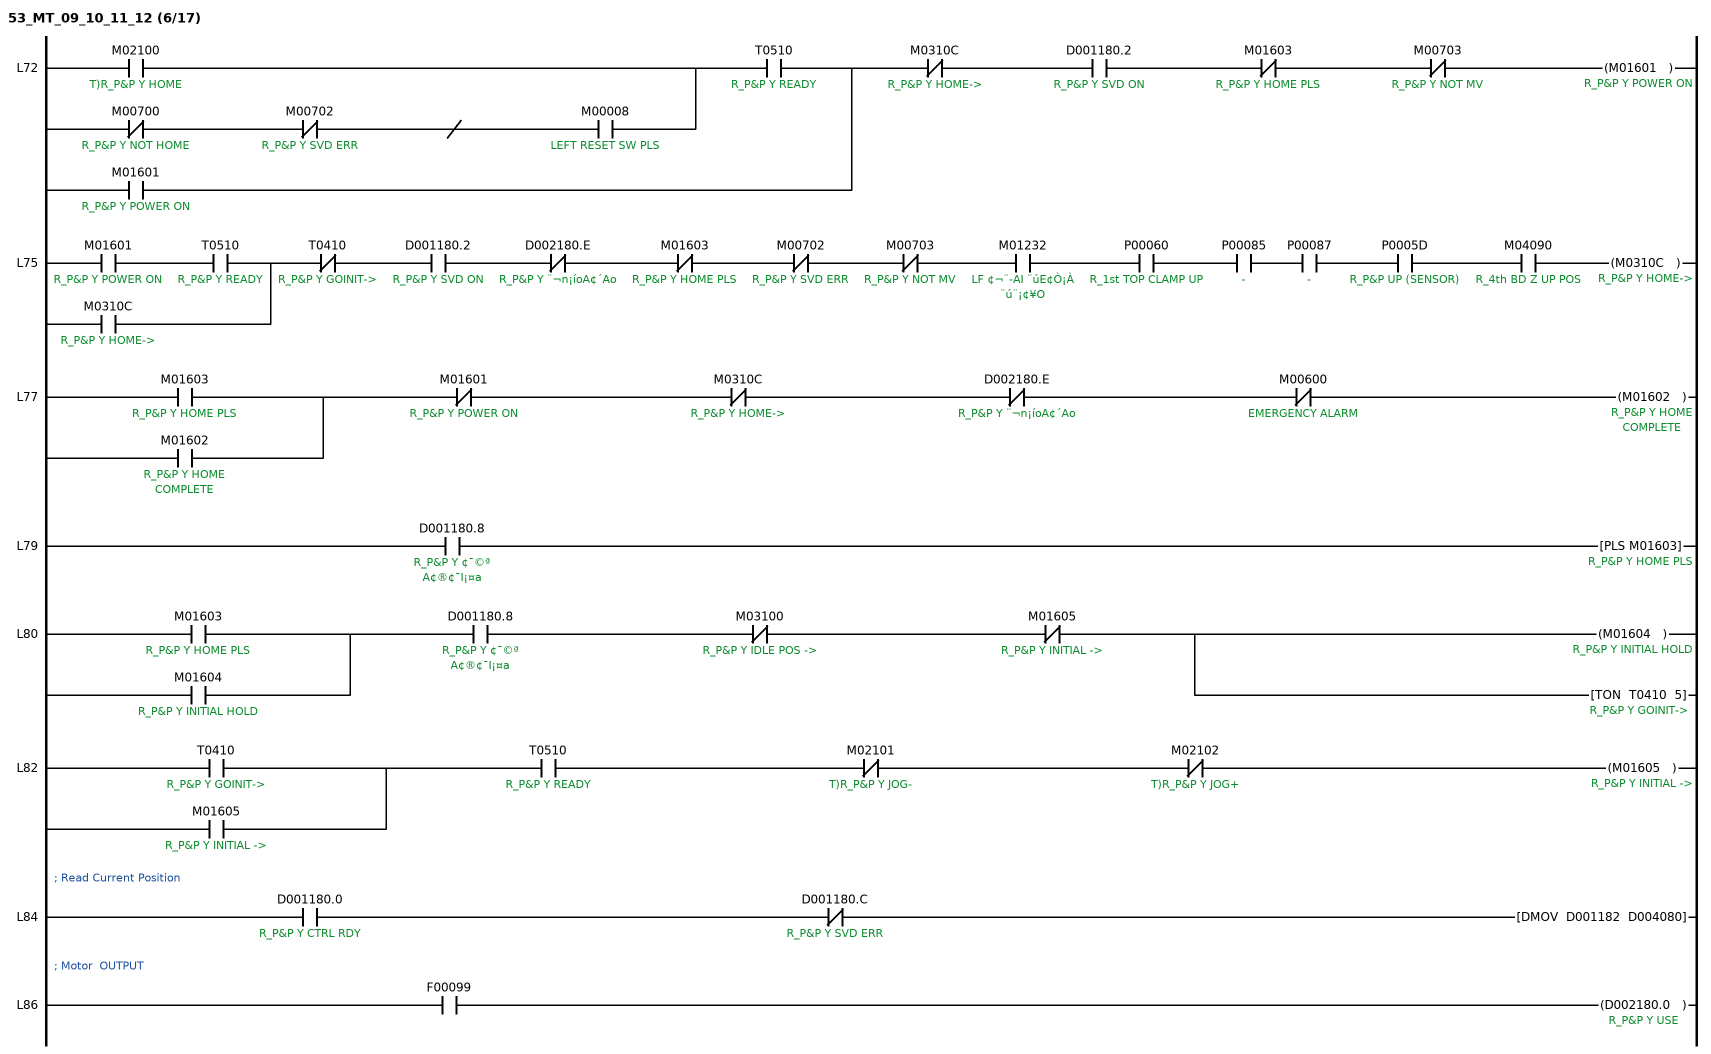
; L72
LOAD      M02100	// T)R_P&P Y HOME
LOAD NOT  M00700	// R_P&P Y NOT HOME
AND NOT   M00702	// R_P&P Y SVD ERR
NOT
AND       M00008	// LEFT RESET SW PLS
OR LOAD
AND       T0510	// R_P&P Y READY
OR        M01601	// R_P&P Y POWER ON
AND NOT   M0310C	// R_P&P Y HOME->
AND       D001180.2	// R_P&P Y SVD ON
AND NOT   M01603	// R_P&P Y HOME PLS
AND NOT   M00703	// R_P&P Y NOT MV
OUT       M01601	// R_P&P Y POWER ON
; L75
LOAD      M01601	// R_P&P Y POWER ON
AND       T0510	// R_P&P Y READY
OR        M0310C	// R_P&P Y HOME->
AND NOT   T0410	// R_P&P Y GOINIT->
AND       D001180.2	// R_P&P Y SVD ON
AND NOT   D002180.E	// R_P&P Y ¨¬n¡íoA¢´Ao
AND NOT   M01603	// R_P&P Y HOME PLS
AND NOT   M00702	// R_P&P Y SVD ERR
AND NOT   M00703	// R_P&P Y NOT MV
AND       M01232	// LF ¢¬¨­AI ¨úE¢Ò¡À ¨ú¨¡¢¥O
AND       P00060	// R_1st TOP CLAMP UP
AND       P00085	// -
AND       P00087	// -
AND       P0005D	// R_P&P UP (SENSOR)
AND       M04090	// R_4th BD Z UP POS
OUT       M0310C	// R_P&P Y HOME->
; L77
LOAD      M01603	// R_P&P Y HOME PLS
OR        M01602	// R_P&P Y HOME COMPLETE
AND NOT   M01601	// R_P&P Y POWER ON
AND NOT   M0310C	// R_P&P Y HOME->
AND NOT   D002180.E	// R_P&P Y ¨¬n¡íoA¢´Ao
AND NOT   M00600	// EMERGENCY ALARM
OUT       M01602	// R_P&P Y HOME COMPLETE
; L79
LOAD      D001180.8	// R_P&P Y ¢¯©ªA¢®¢¯I¡¤a
OUTP      M01603	// R_P&P Y HOME PLS
; L80
LOAD      M01603	// R_P&P Y HOME PLS
OR        M01604	// R_P&P Y INITIAL HOLD
AND       D001180.8	// R_P&P Y ¢¯©ªA¢®¢¯I¡¤a
AND NOT   M03100	// R_P&P Y IDLE POS ->
AND NOT   M01605	// R_P&P Y INITIAL ->
OUT       M01604	// R_P&P Y INITIAL HOLD
TON       T0410 5	// R_P&P Y GOINIT->
; L82
LOAD      T0410	// R_P&P Y GOINIT->
OR        M01605	// R_P&P Y INITIAL ->
AND       T0510	// R_P&P Y READY
AND NOT   M02101	// T)R_P&P Y JOG-
AND NOT   M02102	// T)R_P&P Y JOG+
OUT       M01605	// R_P&P Y INITIAL ->
; L84
LOAD      D001180.0	// R_P&P Y CTRL RDY
AND NOT   D001180.C	// R_P&P Y SVD ERR
DMOV      D001182 D004080
// output comment: Read Current Position
//  Motor  OUTPUT
; L86
LOAD      F00099
OUT       D002180.0	// R_P&P Y USE

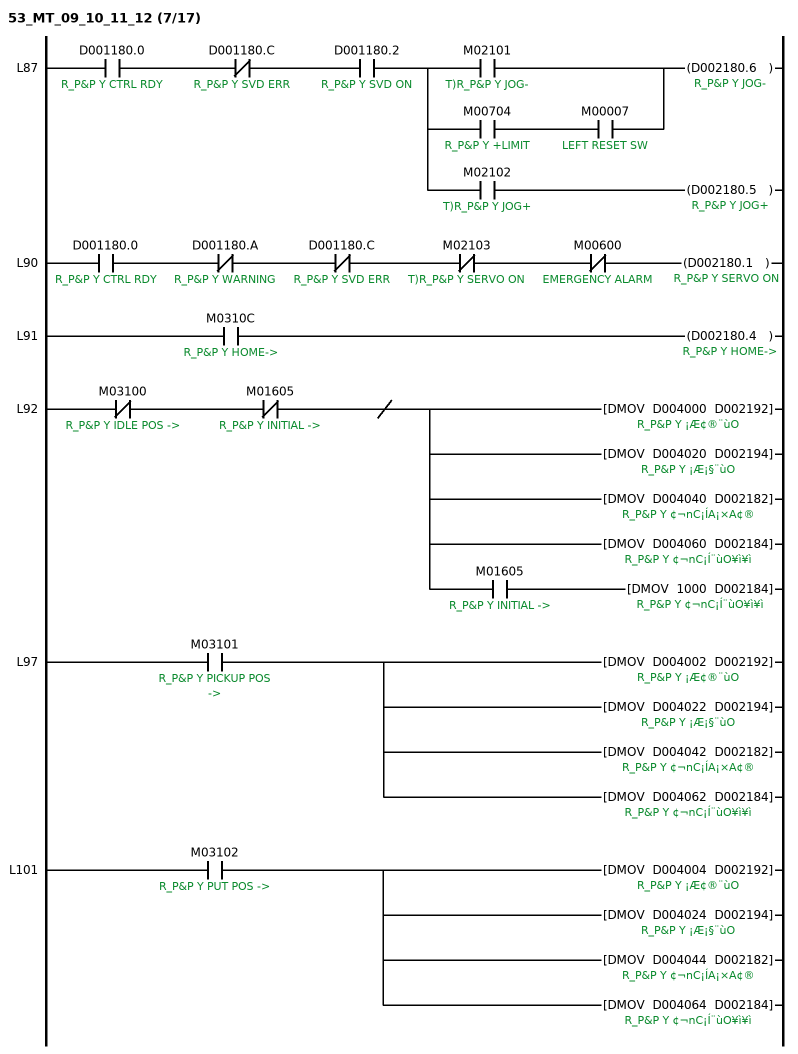
; L87
LOAD      D001180.0	// R_P&P Y CTRL RDY
AND NOT   D001180.C	// R_P&P Y SVD ERR
AND       D001180.2	// R_P&P Y SVD ON
MPUSH
LOAD      M02101	// T)R_P&P Y JOG-
LOAD      M00704	// R_P&P Y +LIMIT
AND       M00007	// LEFT RESET SW
OR LOAD
AND LOAD
OUT       D002180.6	// R_P&P Y JOG-
MPOP
AND       M02102	// T)R_P&P Y JOG+
OUT       D002180.5	// R_P&P Y JOG+
; L90
LOAD      D001180.0	// R_P&P Y CTRL RDY
AND NOT   D001180.A	// R_P&P Y WARNING
AND NOT   D001180.C	// R_P&P Y SVD ERR
AND NOT   M02103	// T)R_P&P Y SERVO ON
AND NOT   M00600	// EMERGENCY ALARM
OUT       D002180.1	// R_P&P Y SERVO ON
; L91
LOAD      M0310C	// R_P&P Y HOME->
OUT       D002180.4	// R_P&P Y HOME->
; L92
LOAD NOT  M03100	// R_P&P Y IDLE POS ->
AND NOT   M01605	// R_P&P Y INITIAL ->
NOT
DMOV      D004000 D002192	// R_P&P Y ¡Æ¢®¨ùO
DMOV      D004020 D002194	// R_P&P Y ¡Æ¡§¨ùO
DMOV      D004040 D002182	// R_P&P Y ¢¬nC¡ÍA¡×A¢®
DMOV      D004060 D002184	// R_P&P Y ¢¬nC¡Í¨ùO¥ì¥ì
AND       M01605	// R_P&P Y INITIAL ->
DMOV      1000 D002184	// R_P&P Y ¢¬nC¡Í¨ùO¥ì¥ì
; L97
LOAD      M03101	// R_P&P Y PICKUP POS ->
DMOV      D004002 D002192	// R_P&P Y ¡Æ¢®¨ùO
DMOV      D004022 D002194	// R_P&P Y ¡Æ¡§¨ùO
DMOV      D004042 D002182	// R_P&P Y ¢¬nC¡ÍA¡×A¢®
DMOV      D004062 D002184	// R_P&P Y ¢¬nC¡Í¨ùO¥ì¥ì
; L101
LOAD      M03102	// R_P&P Y PUT POS ->
DMOV      D004004 D002192	// R_P&P Y ¡Æ¢®¨ùO
DMOV      D004024 D002194	// R_P&P Y ¡Æ¡§¨ùO
DMOV      D004044 D002182	// R_P&P Y ¢¬nC¡ÍA¡×A¢®
DMOV      D004064 D002184	// R_P&P Y ¢¬nC¡Í¨ùO¥ì¥ì

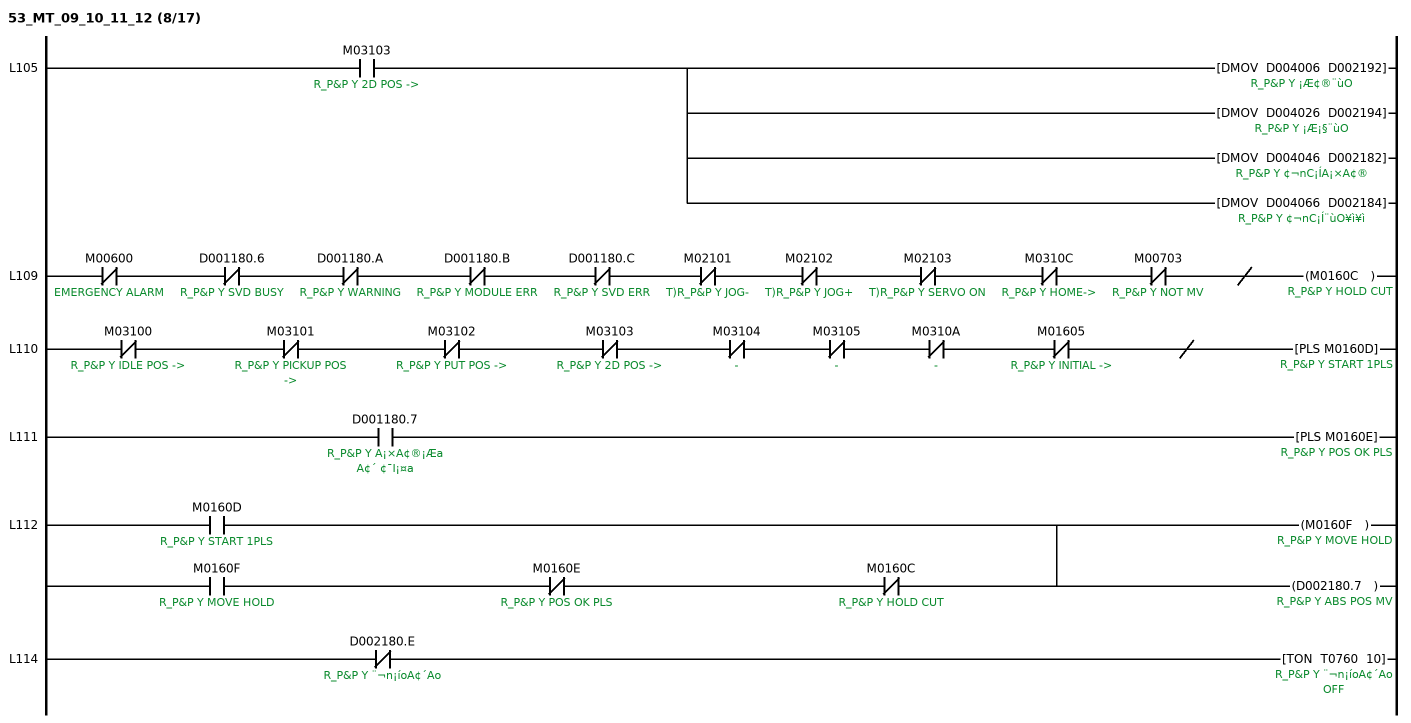
; L105
LOAD      M03103	// R_P&P Y 2D POS ->
DMOV      D004006 D002192	// R_P&P Y ¡Æ¢®¨ùO
DMOV      D004026 D002194	// R_P&P Y ¡Æ¡§¨ùO
DMOV      D004046 D002182	// R_P&P Y ¢¬nC¡ÍA¡×A¢®
DMOV      D004066 D002184	// R_P&P Y ¢¬nC¡Í¨ùO¥ì¥ì
; L109
LOAD NOT  M00600	// EMERGENCY ALARM
AND NOT   D001180.6	// R_P&P Y SVD BUSY
AND NOT   D001180.A	// R_P&P Y WARNING
AND NOT   D001180.B	// R_P&P Y MODULE ERR
AND NOT   D001180.C	// R_P&P Y SVD ERR
AND NOT   M02101	// T)R_P&P Y JOG-
AND NOT   M02102	// T)R_P&P Y JOG+
AND NOT   M02103	// T)R_P&P Y SERVO ON
AND NOT   M0310C	// R_P&P Y HOME->
AND NOT   M00703	// R_P&P Y NOT MV
NOT
OUT       M0160C	// R_P&P Y HOLD CUT
; L110
LOAD NOT  M03100	// R_P&P Y IDLE POS ->
AND NOT   M03101	// R_P&P Y PICKUP POS ->
AND NOT   M03102	// R_P&P Y PUT POS ->
AND NOT   M03103	// R_P&P Y 2D POS ->
AND NOT   M03104	// -
AND NOT   M03105	// -
AND NOT   M0310A	// -
AND NOT   M01605	// R_P&P Y INITIAL ->
NOT
OUTP      M0160D	// R_P&P Y START 1PLS
; L111
LOAD      D001180.7	// R_P&P Y A¡×A¢®¡ÆaA¢´ ¢¯I¡¤a
OUTP      M0160E	// R_P&P Y POS OK PLS
; L112
LOAD      M0160D	// R_P&P Y START 1PLS
LOAD      M0160F	// R_P&P Y MOVE HOLD
AND NOT   M0160E	// R_P&P Y POS OK PLS
AND NOT   M0160C	// R_P&P Y HOLD CUT
OR LOAD
OUT       M0160F	// R_P&P Y MOVE HOLD
OUT       D002180.7	// R_P&P Y ABS POS MV
; L114
LOAD NOT  D002180.E	// R_P&P Y ¨¬n¡íoA¢´Ao
TON       T0760 10	// R_P&P Y ¨¬n¡íoA¢´AoOFF

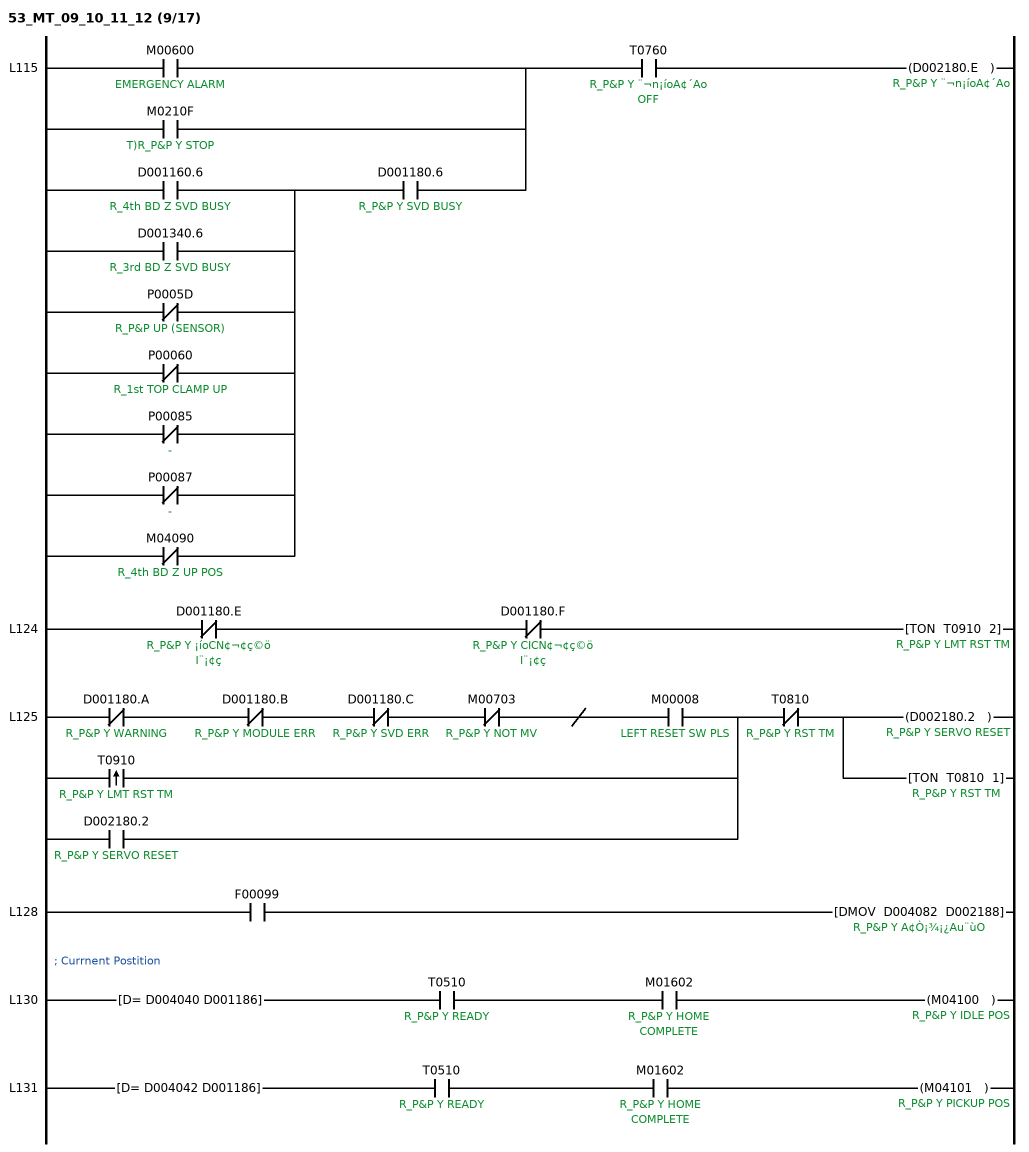
; L115
LOAD      M00600	// EMERGENCY ALARM
OR        M0210F	// T)R_P&P Y STOP
LOAD      D001160.6	// R_4th BD Z SVD BUSY
OR        D001340.6	// R_3rd BD Z SVD BUSY
OR NOT    P0005D	// R_P&P UP (SENSOR)
OR NOT    P00060	// R_1st TOP CLAMP UP
OR NOT    P00085	// -
OR NOT    P00087	// -
OR NOT    M04090	// R_4th BD Z UP POS
AND       D001180.6	// R_P&P Y SVD BUSY
OR LOAD
AND       T0760	// R_P&P Y ¨¬n¡íoA¢´AoOFF
OUT       D002180.E	// R_P&P Y ¨¬n¡íoA¢´Ao
; L124
LOAD NOT  D001180.E	// R_P&P Y ¡íoCN¢¬¢ç©öI¨¡¢ç
AND NOT   D001180.F	// R_P&P Y CICN¢¬¢ç©öI¨¡¢ç
TON       T0910 2	// R_P&P Y LMT RST TM
; L125
LOAD NOT  D001180.A	// R_P&P Y WARNING
AND NOT   D001180.B	// R_P&P Y MODULE ERR
AND NOT   D001180.C	// R_P&P Y SVD ERR
AND NOT   M00703	// R_P&P Y NOT MV
NOT
AND       M00008	// LEFT RESET SW PLS
ORP       T0910	// R_P&P Y LMT RST TM
OR        D002180.2	// R_P&P Y SERVO RESET
AND NOT   T0810	// R_P&P Y RST TM
OUT       D002180.2	// R_P&P Y SERVO RESET
TON       T0810 1	// R_P&P Y RST TM
; L128
LOAD      F00099
DMOV      D004082 D002188	// R_P&P Y A¢Ò¡¾¡¿Au¨ùO
// Currnent Postition
; L130
LOADD=    D004040 D001186
AND       T0510	// R_P&P Y READY
AND       M01602	// R_P&P Y HOME COMPLETE
OUT       M04100	// R_P&P Y IDLE POS
; L131
LOADD=    D004042 D001186
AND       T0510	// R_P&P Y READY
AND       M01602	// R_P&P Y HOME COMPLETE
OUT       M04101	// R_P&P Y PICKUP POS

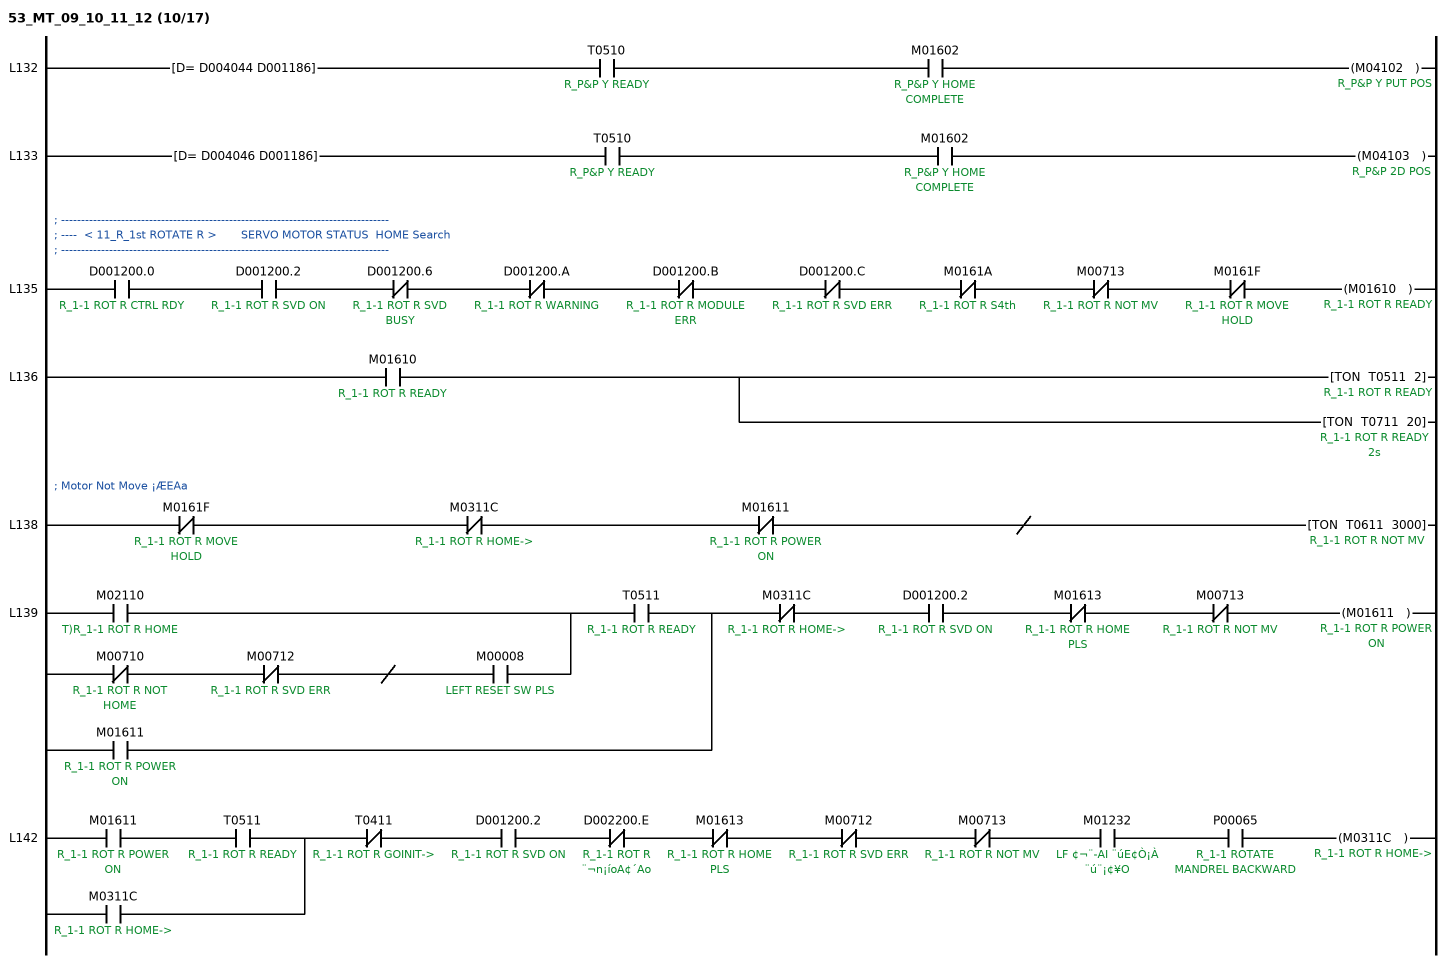
; L132
LOADD=    D004044 D001186
AND       T0510	// R_P&P Y READY
AND       M01602	// R_P&P Y HOME COMPLETE
OUT       M04102	// R_P&P Y PUT POS
; L133
LOADD=    D004046 D001186
AND       T0510	// R_P&P Y READY
AND       M01602	// R_P&P Y HOME COMPLETE
OUT       M04103	// R_P&P 2D POS
// ----------------------------------------------------------------------------------
// 
// ----  < 11_R_1st ROTATE R >       SERVO MOTOR STATUS  HOME Search
// 
// ----------------------------------------------------------------------------------
; L135
LOAD      D001200.0	// R_1-1 ROT R CTRL RDY
AND       D001200.2	// R_1-1 ROT R SVD ON
AND NOT   D001200.6	// R_1-1 ROT R SVD BUSY
AND NOT   D001200.A	// R_1-1 ROT R WARNING
AND NOT   D001200.B	// R_1-1 ROT R MODULE ERR
AND NOT   D001200.C	// R_1-1 ROT R SVD ERR
AND NOT   M0161A	// R_1-1 ROT R S4th
AND NOT   M00713	// R_1-1 ROT R NOT MV
AND NOT   M0161F	// R_1-1 ROT R MOVE HOLD
OUT       M01610	// R_1-1 ROT R READY
; L136
LOAD      M01610	// R_1-1 ROT R READY
TON       T0511 2	// R_1-1 ROT R READY
TON       T0711 20	// R_1-1 ROT R READY 2s
; L138
LOAD NOT  M0161F	// R_1-1 ROT R MOVE HOLD
AND NOT   M0311C	// R_1-1 ROT R HOME->
AND NOT   M01611	// R_1-1 ROT R POWER ON
NOT
TON       T0611 3000	// R_1-1 ROT R NOT MV
// output comment: Motor Not Move ¡ÆEAa
; L139
LOAD      M02110	// T)R_1-1 ROT R HOME
LOAD NOT  M00710	// R_1-1 ROT R NOT HOME
AND NOT   M00712	// R_1-1 ROT R SVD ERR
NOT
AND       M00008	// LEFT RESET SW PLS
OR LOAD
AND       T0511	// R_1-1 ROT R READY
OR        M01611	// R_1-1 ROT R POWER ON
AND NOT   M0311C	// R_1-1 ROT R HOME->
AND       D001200.2	// R_1-1 ROT R SVD ON
AND NOT   M01613	// R_1-1 ROT R HOME PLS
AND NOT   M00713	// R_1-1 ROT R NOT MV
OUT       M01611	// R_1-1 ROT R POWER ON
; L142
LOAD      M01611	// R_1-1 ROT R POWER ON
AND       T0511	// R_1-1 ROT R READY
OR        M0311C	// R_1-1 ROT R HOME->
AND NOT   T0411	// R_1-1 ROT R GOINIT->
AND       D001200.2	// R_1-1 ROT R SVD ON
AND NOT   D002200.E	// R_1-1 ROT R ¨¬n¡íoA¢´Ao
AND NOT   M01613	// R_1-1 ROT R HOME PLS
AND NOT   M00712	// R_1-1 ROT R SVD ERR
AND NOT   M00713	// R_1-1 ROT R NOT MV
AND       M01232	// LF ¢¬¨­AI ¨úE¢Ò¡À ¨ú¨¡¢¥O
AND       P00065	// R_1-1 ROTATE MANDREL BACKWARD
OUT       M0311C	// R_1-1 ROT R HOME->

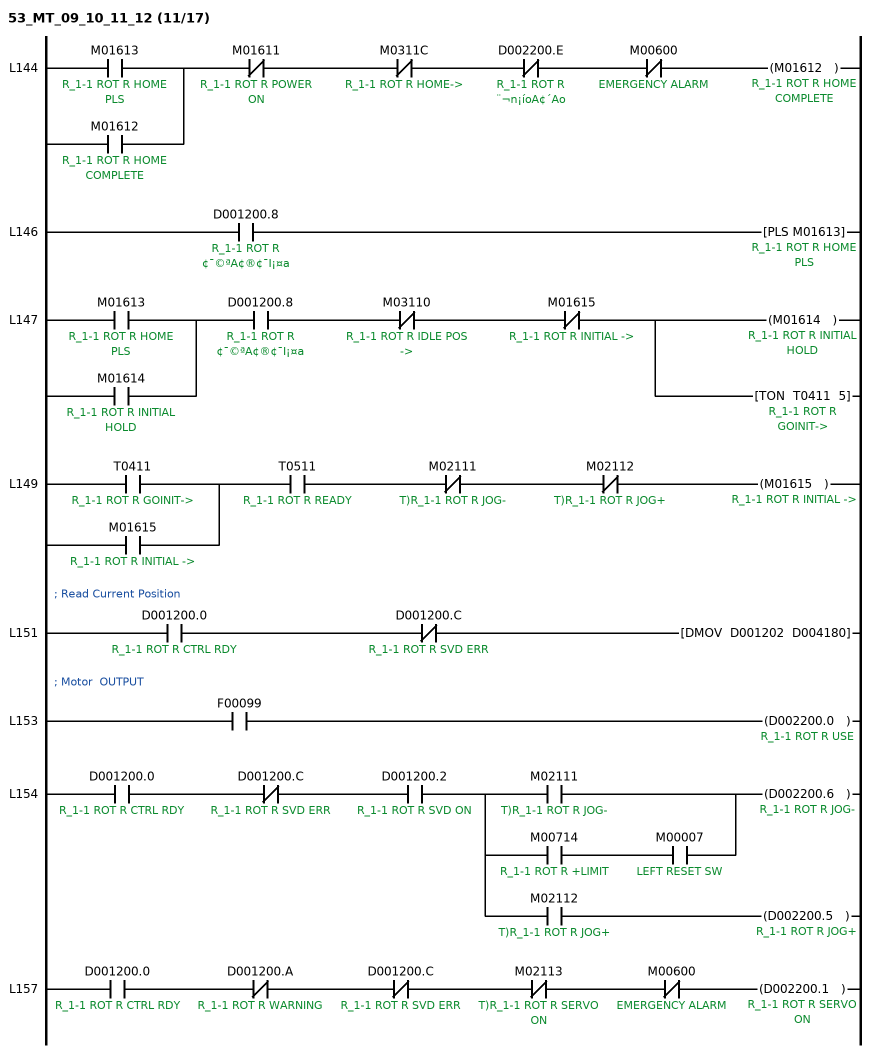
; L144
LOAD      M01613	// R_1-1 ROT R HOME PLS
OR        M01612	// R_1-1 ROT R HOME COMPLETE
AND NOT   M01611	// R_1-1 ROT R POWER ON
AND NOT   M0311C	// R_1-1 ROT R HOME->
AND NOT   D002200.E	// R_1-1 ROT R ¨¬n¡íoA¢´Ao
AND NOT   M00600	// EMERGENCY ALARM
OUT       M01612	// R_1-1 ROT R HOME COMPLETE
; L146
LOAD      D001200.8	// R_1-1 ROT R ¢¯©ªA¢®¢¯I¡¤a
OUTP      M01613	// R_1-1 ROT R HOME PLS
; L147
LOAD      M01613	// R_1-1 ROT R HOME PLS
OR        M01614	// R_1-1 ROT R INITIAL HOLD
AND       D001200.8	// R_1-1 ROT R ¢¯©ªA¢®¢¯I¡¤a
AND NOT   M03110	// R_1-1 ROT R IDLE POS ->
AND NOT   M01615	// R_1-1 ROT R INITIAL ->
OUT       M01614	// R_1-1 ROT R INITIAL HOLD
TON       T0411 5	// R_1-1 ROT R GOINIT->
; L149
LOAD      T0411	// R_1-1 ROT R GOINIT->
OR        M01615	// R_1-1 ROT R INITIAL ->
AND       T0511	// R_1-1 ROT R READY
AND NOT   M02111	// T)R_1-1 ROT R JOG-
AND NOT   M02112	// T)R_1-1 ROT R JOG+
OUT       M01615	// R_1-1 ROT R INITIAL ->
; L151
LOAD      D001200.0	// R_1-1 ROT R CTRL RDY
AND NOT   D001200.C	// R_1-1 ROT R SVD ERR
DMOV      D001202 D004180
// output comment: Read Current Position
//  Motor  OUTPUT
; L153
LOAD      F00099
OUT       D002200.0	// R_1-1 ROT R USE
; L154
LOAD      D001200.0	// R_1-1 ROT R CTRL RDY
AND NOT   D001200.C	// R_1-1 ROT R SVD ERR
AND       D001200.2	// R_1-1 ROT R SVD ON
MPUSH
LOAD      M02111	// T)R_1-1 ROT R JOG-
LOAD      M00714	// R_1-1 ROT R +LIMIT
AND       M00007	// LEFT RESET SW
OR LOAD
AND LOAD
OUT       D002200.6	// R_1-1 ROT R JOG-
MPOP
AND       M02112	// T)R_1-1 ROT R JOG+
OUT       D002200.5	// R_1-1 ROT R JOG+
; L157
LOAD      D001200.0	// R_1-1 ROT R CTRL RDY
AND NOT   D001200.A	// R_1-1 ROT R WARNING
AND NOT   D001200.C	// R_1-1 ROT R SVD ERR
AND NOT   M02113	// T)R_1-1 ROT R SERVO ON
AND NOT   M00600	// EMERGENCY ALARM
OUT       D002200.1	// R_1-1 ROT R SERVO ON

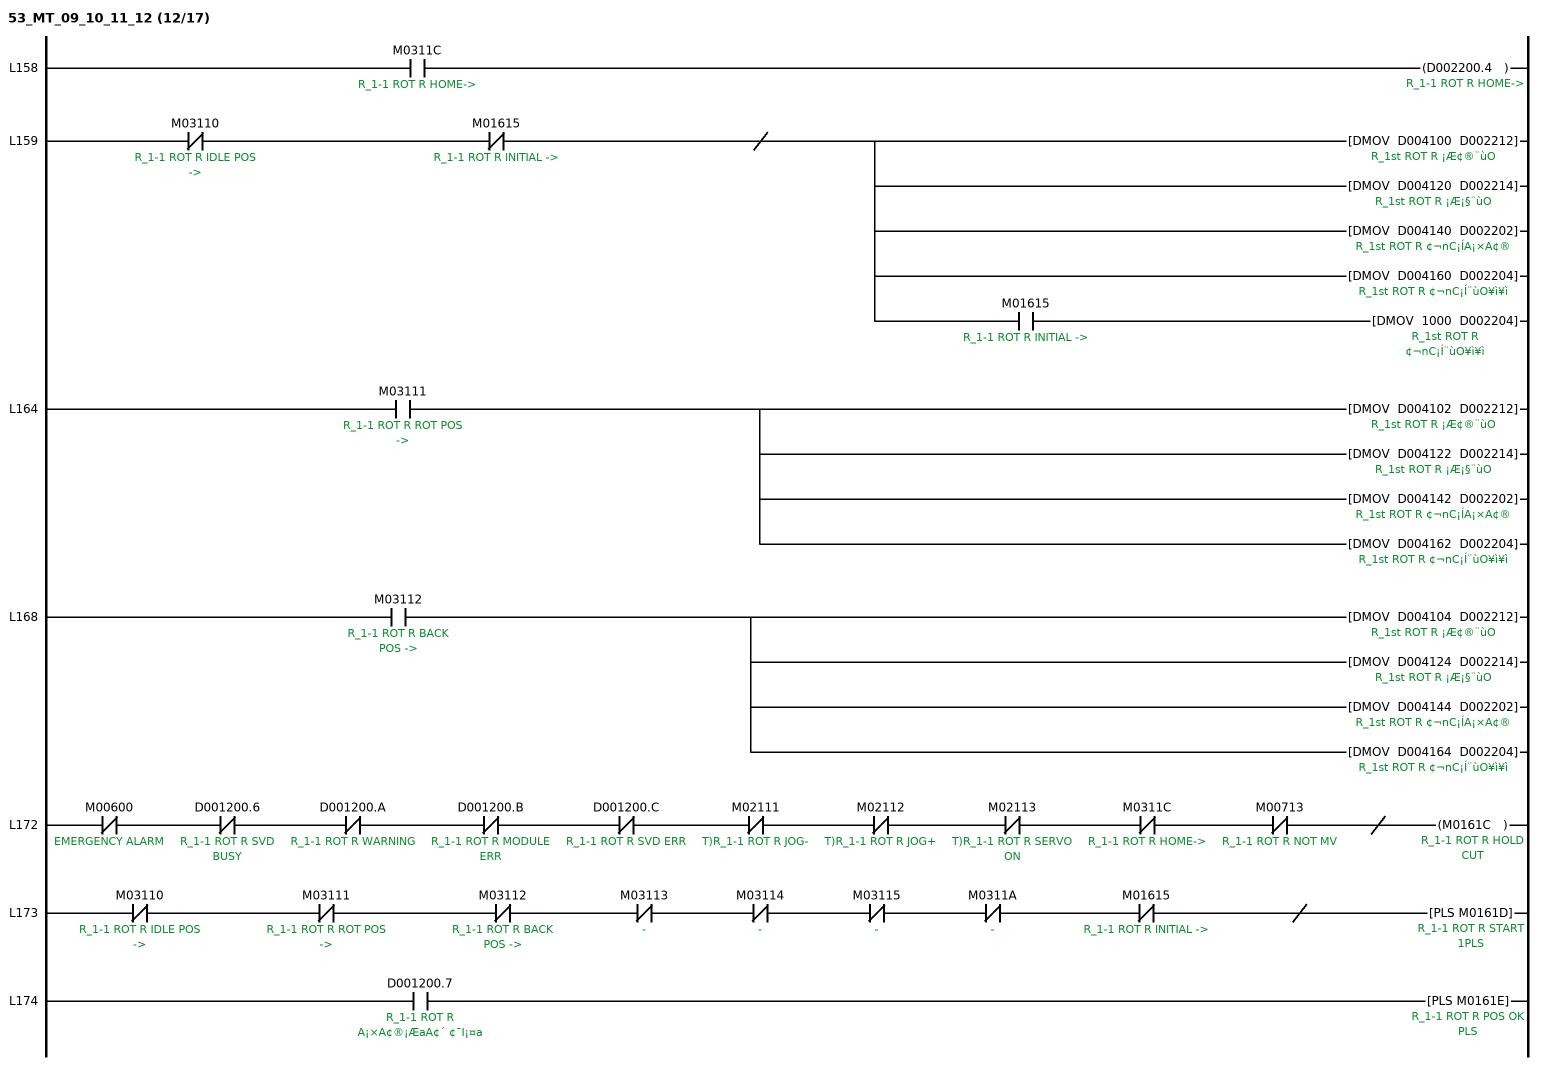
; L158
LOAD      M0311C	// R_1-1 ROT R HOME->
OUT       D002200.4	// R_1-1 ROT R HOME->
; L159
LOAD NOT  M03110	// R_1-1 ROT R IDLE POS ->
AND NOT   M01615	// R_1-1 ROT R INITIAL ->
NOT
DMOV      D004100 D002212	// R_1st ROT R ¡Æ¢®¨ùO
DMOV      D004120 D002214	// R_1st ROT R ¡Æ¡§¨ùO
DMOV      D004140 D002202	// R_1st ROT R ¢¬nC¡ÍA¡×A¢®
DMOV      D004160 D002204	// R_1st ROT R ¢¬nC¡Í¨ùO¥ì¥ì
AND       M01615	// R_1-1 ROT R INITIAL ->
DMOV      1000 D002204	// R_1st ROT R ¢¬nC¡Í¨ùO¥ì¥ì
; L164
LOAD      M03111	// R_1-1 ROT R ROT POS ->
DMOV      D004102 D002212	// R_1st ROT R ¡Æ¢®¨ùO
DMOV      D004122 D002214	// R_1st ROT R ¡Æ¡§¨ùO
DMOV      D004142 D002202	// R_1st ROT R ¢¬nC¡ÍA¡×A¢®
DMOV      D004162 D002204	// R_1st ROT R ¢¬nC¡Í¨ùO¥ì¥ì
; L168
LOAD      M03112	// R_1-1 ROT R BACK POS ->
DMOV      D004104 D002212	// R_1st ROT R ¡Æ¢®¨ùO
DMOV      D004124 D002214	// R_1st ROT R ¡Æ¡§¨ùO
DMOV      D004144 D002202	// R_1st ROT R ¢¬nC¡ÍA¡×A¢®
DMOV      D004164 D002204	// R_1st ROT R ¢¬nC¡Í¨ùO¥ì¥ì
; L172
LOAD NOT  M00600	// EMERGENCY ALARM
AND NOT   D001200.6	// R_1-1 ROT R SVD BUSY
AND NOT   D001200.A	// R_1-1 ROT R WARNING
AND NOT   D001200.B	// R_1-1 ROT R MODULE ERR
AND NOT   D001200.C	// R_1-1 ROT R SVD ERR
AND NOT   M02111	// T)R_1-1 ROT R JOG-
AND NOT   M02112	// T)R_1-1 ROT R JOG+
AND NOT   M02113	// T)R_1-1 ROT R SERVO ON
AND NOT   M0311C	// R_1-1 ROT R HOME->
AND NOT   M00713	// R_1-1 ROT R NOT MV
NOT
OUT       M0161C	// R_1-1 ROT R HOLD CUT
; L173
LOAD NOT  M03110	// R_1-1 ROT R IDLE POS ->
AND NOT   M03111	// R_1-1 ROT R ROT POS ->
AND NOT   M03112	// R_1-1 ROT R BACK POS ->
AND NOT   M03113	// -
AND NOT   M03114	// -
AND NOT   M03115	// -
AND NOT   M0311A	// -
AND NOT   M01615	// R_1-1 ROT R INITIAL ->
NOT
OUTP      M0161D	// R_1-1 ROT R START 1PLS
; L174
LOAD      D001200.7	// R_1-1 ROT R A¡×A¢®¡ÆaA¢´ ¢¯I¡¤a
OUTP      M0161E	// R_1-1 ROT R POS OK PLS

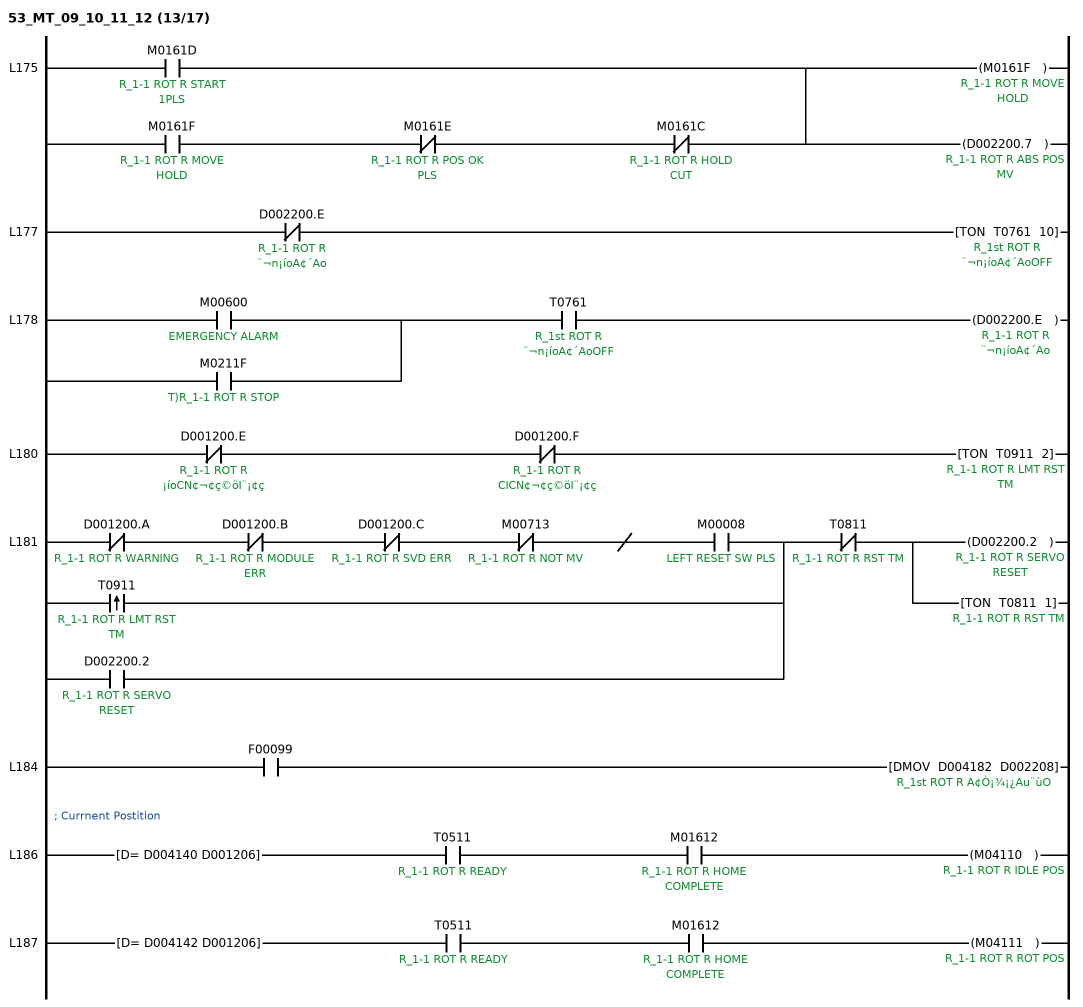
; L175
LOAD      M0161D	// R_1-1 ROT R START 1PLS
LOAD      M0161F	// R_1-1 ROT R MOVE HOLD
AND NOT   M0161E	// R_1-1 ROT R POS OK PLS
AND NOT   M0161C	// R_1-1 ROT R HOLD CUT
OR LOAD
OUT       M0161F	// R_1-1 ROT R MOVE HOLD
OUT       D002200.7	// R_1-1 ROT R ABS POS MV
; L177
LOAD NOT  D002200.E	// R_1-1 ROT R ¨¬n¡íoA¢´Ao
TON       T0761 10	// R_1st ROT R ¨¬n¡íoA¢´AoOFF
; L178
LOAD      M00600	// EMERGENCY ALARM
OR        M0211F	// T)R_1-1 ROT R STOP
AND       T0761	// R_1st ROT R ¨¬n¡íoA¢´AoOFF
OUT       D002200.E	// R_1-1 ROT R ¨¬n¡íoA¢´Ao
; L180
LOAD NOT  D001200.E	// R_1-1 ROT R ¡íoCN¢¬¢ç©öI¨¡¢ç
AND NOT   D001200.F	// R_1-1 ROT R CICN¢¬¢ç©öI¨¡¢ç
TON       T0911 2	// R_1-1 ROT R LMT RST TM
; L181
LOAD NOT  D001200.A	// R_1-1 ROT R WARNING
AND NOT   D001200.B	// R_1-1 ROT R MODULE ERR
AND NOT   D001200.C	// R_1-1 ROT R SVD ERR
AND NOT   M00713	// R_1-1 ROT R NOT MV
NOT
AND       M00008	// LEFT RESET SW PLS
ORP       T0911	// R_1-1 ROT R LMT RST TM
OR        D002200.2	// R_1-1 ROT R SERVO RESET
AND NOT   T0811	// R_1-1 ROT R RST TM
OUT       D002200.2	// R_1-1 ROT R SERVO RESET
TON       T0811 1	// R_1-1 ROT R RST TM
; L184
LOAD      F00099
DMOV      D004182 D002208	// R_1st ROT R A¢Ò¡¾¡¿Au¨ùO
// Currnent Postition
; L186
LOADD=    D004140 D001206
AND       T0511	// R_1-1 ROT R READY
AND       M01612	// R_1-1 ROT R HOME COMPLETE
OUT       M04110	// R_1-1 ROT R IDLE POS
; L187
LOADD=    D004142 D001206
AND       T0511	// R_1-1 ROT R READY
AND       M01612	// R_1-1 ROT R HOME COMPLETE
OUT       M04111	// R_1-1 ROT R ROT POS

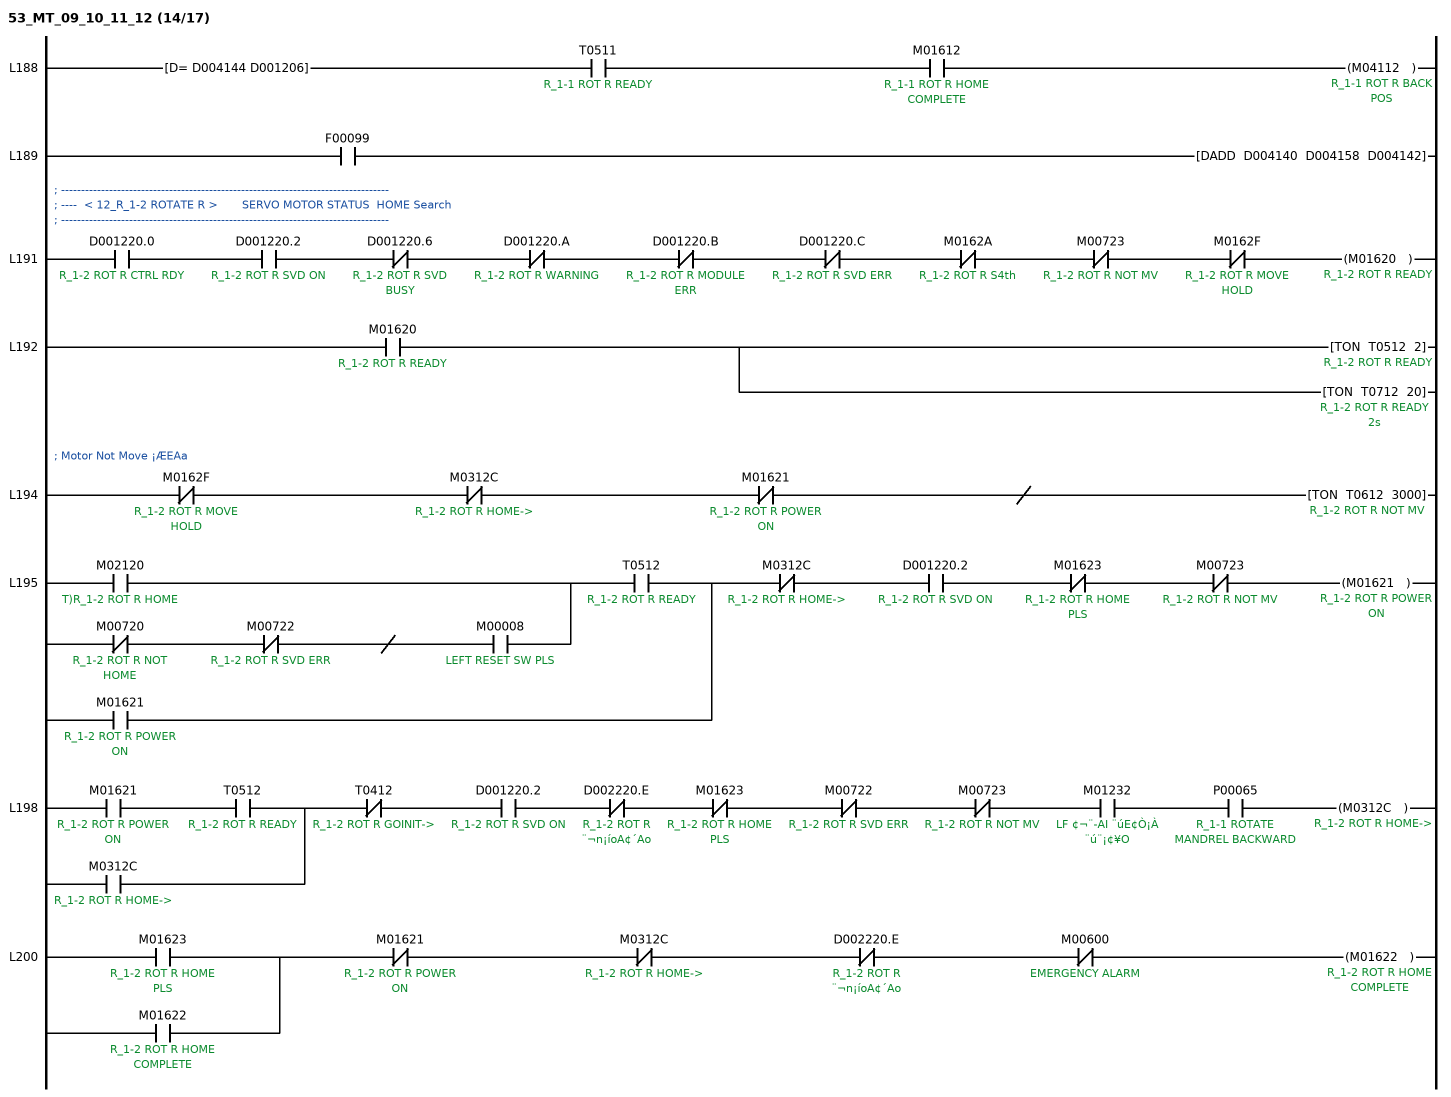
; L188
LOADD=    D004144 D001206
AND       T0511	// R_1-1 ROT R READY
AND       M01612	// R_1-1 ROT R HOME COMPLETE
OUT       M04112	// R_1-1 ROT R BACK POS
; L189
LOAD      F00099
DADD      D004140 D004158 D004142
// ----------------------------------------------------------------------------------
// 
// ----  < 12_R_1-2 ROTATE R >       SERVO MOTOR STATUS  HOME Search
// 
// ----------------------------------------------------------------------------------
; L191
LOAD      D001220.0	// R_1-2 ROT R CTRL RDY
AND       D001220.2	// R_1-2 ROT R SVD ON
AND NOT   D001220.6	// R_1-2 ROT R SVD BUSY
AND NOT   D001220.A	// R_1-2 ROT R WARNING
AND NOT   D001220.B	// R_1-2 ROT R MODULE ERR
AND NOT   D001220.C	// R_1-2 ROT R SVD ERR
AND NOT   M0162A	// R_1-2 ROT R S4th
AND NOT   M00723	// R_1-2 ROT R NOT MV
AND NOT   M0162F	// R_1-2 ROT R MOVE HOLD
OUT       M01620	// R_1-2 ROT R READY
; L192
LOAD      M01620	// R_1-2 ROT R READY
TON       T0512 2	// R_1-2 ROT R READY
TON       T0712 20	// R_1-2 ROT R READY 2s
; L194
LOAD NOT  M0162F	// R_1-2 ROT R MOVE HOLD
AND NOT   M0312C	// R_1-2 ROT R HOME->
AND NOT   M01621	// R_1-2 ROT R POWER ON
NOT
TON       T0612 3000	// R_1-2 ROT R NOT MV
// output comment: Motor Not Move ¡ÆEAa
; L195
LOAD      M02120	// T)R_1-2 ROT R HOME
LOAD NOT  M00720	// R_1-2 ROT R NOT HOME
AND NOT   M00722	// R_1-2 ROT R SVD ERR
NOT
AND       M00008	// LEFT RESET SW PLS
OR LOAD
AND       T0512	// R_1-2 ROT R READY
OR        M01621	// R_1-2 ROT R POWER ON
AND NOT   M0312C	// R_1-2 ROT R HOME->
AND       D001220.2	// R_1-2 ROT R SVD ON
AND NOT   M01623	// R_1-2 ROT R HOME PLS
AND NOT   M00723	// R_1-2 ROT R NOT MV
OUT       M01621	// R_1-2 ROT R POWER ON
; L198
LOAD      M01621	// R_1-2 ROT R POWER ON
AND       T0512	// R_1-2 ROT R READY
OR        M0312C	// R_1-2 ROT R HOME->
AND NOT   T0412	// R_1-2 ROT R GOINIT->
AND       D001220.2	// R_1-2 ROT R SVD ON
AND NOT   D002220.E	// R_1-2 ROT R ¨¬n¡íoA¢´Ao
AND NOT   M01623	// R_1-2 ROT R HOME PLS
AND NOT   M00722	// R_1-2 ROT R SVD ERR
AND NOT   M00723	// R_1-2 ROT R NOT MV
AND       M01232	// LF ¢¬¨­AI ¨úE¢Ò¡À ¨ú¨¡¢¥O
AND       P00065	// R_1-1 ROTATE MANDREL BACKWARD
OUT       M0312C	// R_1-2 ROT R HOME->
; L200
LOAD      M01623	// R_1-2 ROT R HOME PLS
OR        M01622	// R_1-2 ROT R HOME COMPLETE
AND NOT   M01621	// R_1-2 ROT R POWER ON
AND NOT   M0312C	// R_1-2 ROT R HOME->
AND NOT   D002220.E	// R_1-2 ROT R ¨¬n¡íoA¢´Ao
AND NOT   M00600	// EMERGENCY ALARM
OUT       M01622	// R_1-2 ROT R HOME COMPLETE

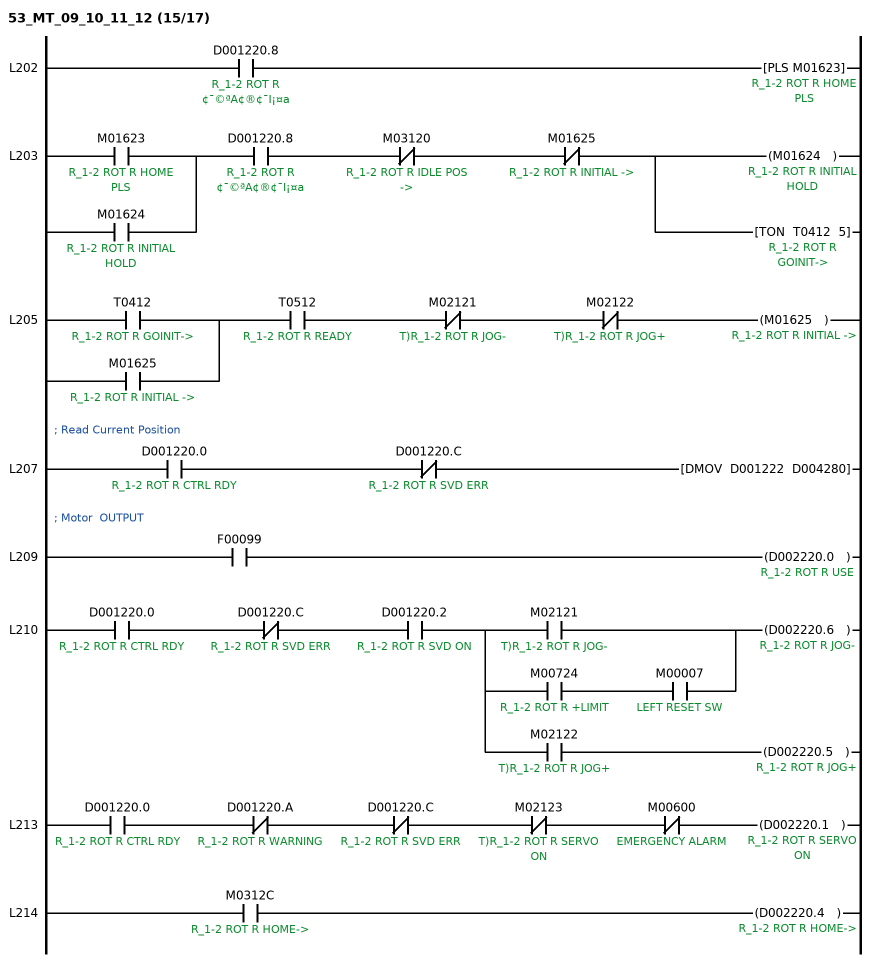
; L202
LOAD      D001220.8	// R_1-2 ROT R ¢¯©ªA¢®¢¯I¡¤a
OUTP      M01623	// R_1-2 ROT R HOME PLS
; L203
LOAD      M01623	// R_1-2 ROT R HOME PLS
OR        M01624	// R_1-2 ROT R INITIAL HOLD
AND       D001220.8	// R_1-2 ROT R ¢¯©ªA¢®¢¯I¡¤a
AND NOT   M03120	// R_1-2 ROT R IDLE POS ->
AND NOT   M01625	// R_1-2 ROT R INITIAL ->
OUT       M01624	// R_1-2 ROT R INITIAL HOLD
TON       T0412 5	// R_1-2 ROT R GOINIT->
; L205
LOAD      T0412	// R_1-2 ROT R GOINIT->
OR        M01625	// R_1-2 ROT R INITIAL ->
AND       T0512	// R_1-2 ROT R READY
AND NOT   M02121	// T)R_1-2 ROT R JOG-
AND NOT   M02122	// T)R_1-2 ROT R JOG+
OUT       M01625	// R_1-2 ROT R INITIAL ->
; L207
LOAD      D001220.0	// R_1-2 ROT R CTRL RDY
AND NOT   D001220.C	// R_1-2 ROT R SVD ERR
DMOV      D001222 D004280
// output comment: Read Current Position
//  Motor  OUTPUT
; L209
LOAD      F00099
OUT       D002220.0	// R_1-2 ROT R USE
; L210
LOAD      D001220.0	// R_1-2 ROT R CTRL RDY
AND NOT   D001220.C	// R_1-2 ROT R SVD ERR
AND       D001220.2	// R_1-2 ROT R SVD ON
MPUSH
LOAD      M02121	// T)R_1-2 ROT R JOG-
LOAD      M00724	// R_1-2 ROT R +LIMIT
AND       M00007	// LEFT RESET SW
OR LOAD
AND LOAD
OUT       D002220.6	// R_1-2 ROT R JOG-
MPOP
AND       M02122	// T)R_1-2 ROT R JOG+
OUT       D002220.5	// R_1-2 ROT R JOG+
; L213
LOAD      D001220.0	// R_1-2 ROT R CTRL RDY
AND NOT   D001220.A	// R_1-2 ROT R WARNING
AND NOT   D001220.C	// R_1-2 ROT R SVD ERR
AND NOT   M02123	// T)R_1-2 ROT R SERVO ON
AND NOT   M00600	// EMERGENCY ALARM
OUT       D002220.1	// R_1-2 ROT R SERVO ON
; L214
LOAD      M0312C	// R_1-2 ROT R HOME->
OUT       D002220.4	// R_1-2 ROT R HOME->

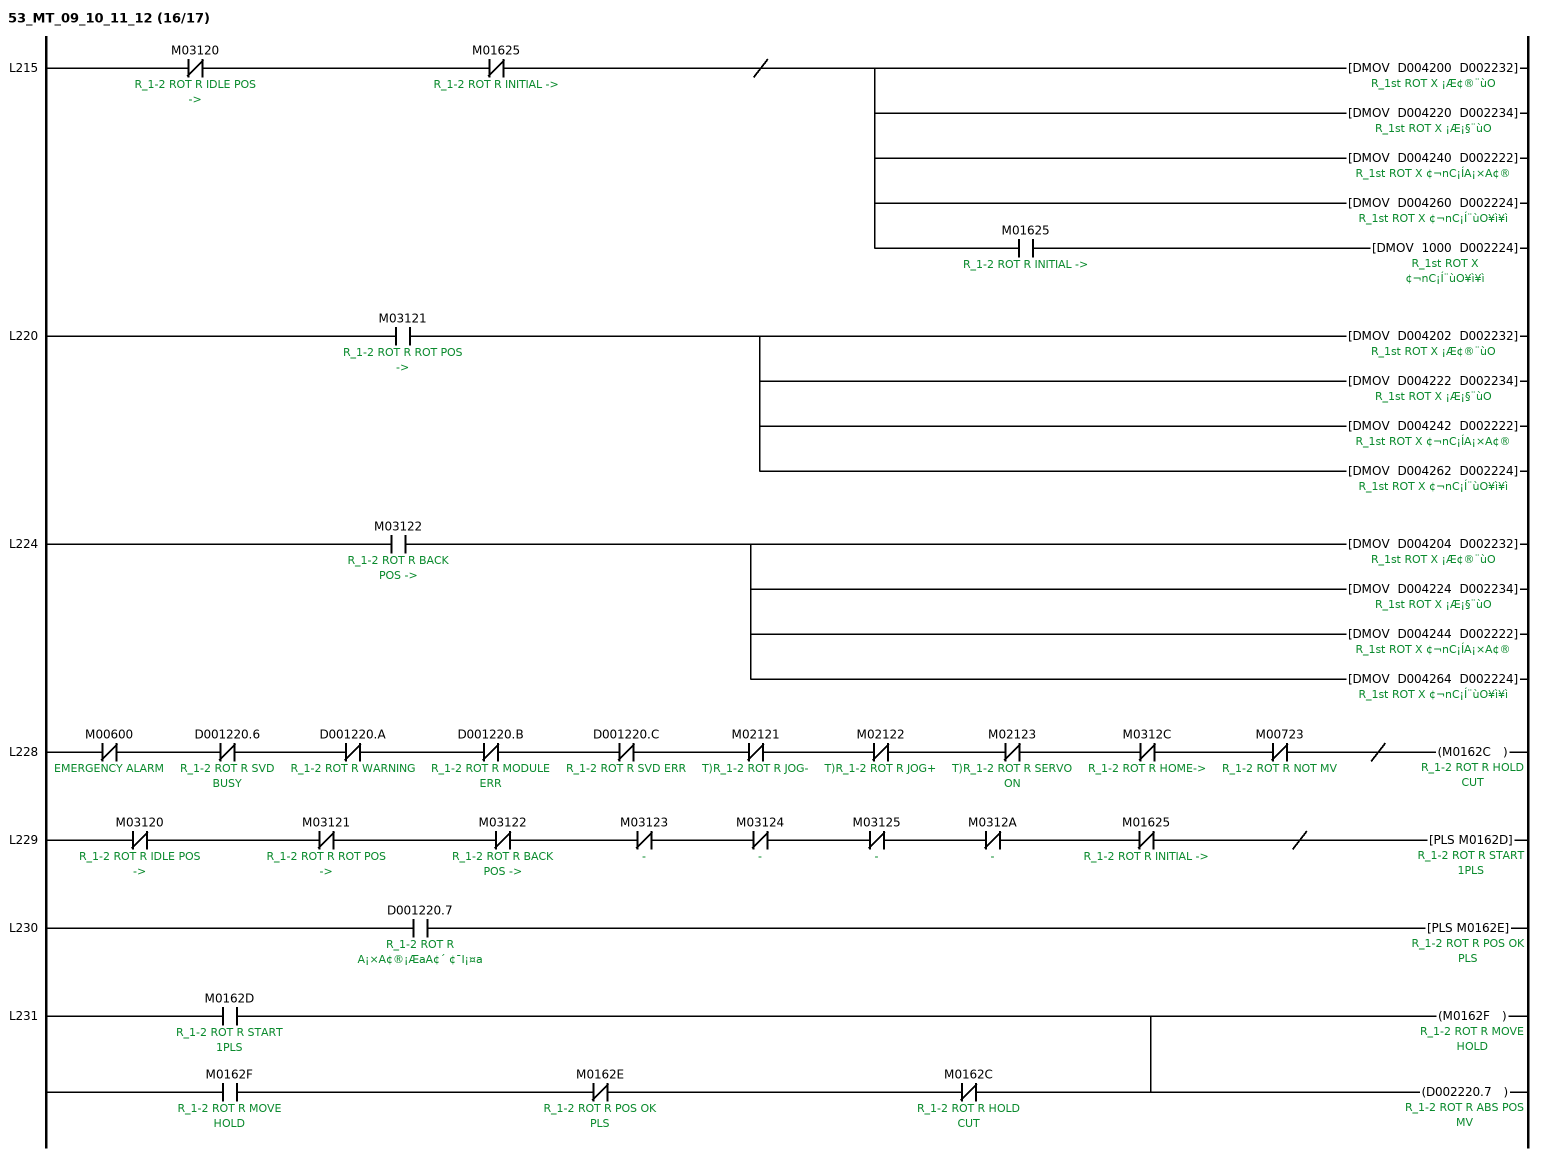
; L215
LOAD NOT  M03120	// R_1-2 ROT R IDLE POS ->
AND NOT   M01625	// R_1-2 ROT R INITIAL ->
NOT
DMOV      D004200 D002232	// R_1st ROT X ¡Æ¢®¨ùO
DMOV      D004220 D002234	// R_1st ROT X ¡Æ¡§¨ùO
DMOV      D004240 D002222	// R_1st ROT X ¢¬nC¡ÍA¡×A¢®
DMOV      D004260 D002224	// R_1st ROT X ¢¬nC¡Í¨ùO¥ì¥ì
AND       M01625	// R_1-2 ROT R INITIAL ->
DMOV      1000 D002224	// R_1st ROT X ¢¬nC¡Í¨ùO¥ì¥ì
; L220
LOAD      M03121	// R_1-2 ROT R ROT POS ->
DMOV      D004202 D002232	// R_1st ROT X ¡Æ¢®¨ùO
DMOV      D004222 D002234	// R_1st ROT X ¡Æ¡§¨ùO
DMOV      D004242 D002222	// R_1st ROT X ¢¬nC¡ÍA¡×A¢®
DMOV      D004262 D002224	// R_1st ROT X ¢¬nC¡Í¨ùO¥ì¥ì
; L224
LOAD      M03122	// R_1-2 ROT R BACK POS ->
DMOV      D004204 D002232	// R_1st ROT X ¡Æ¢®¨ùO
DMOV      D004224 D002234	// R_1st ROT X ¡Æ¡§¨ùO
DMOV      D004244 D002222	// R_1st ROT X ¢¬nC¡ÍA¡×A¢®
DMOV      D004264 D002224	// R_1st ROT X ¢¬nC¡Í¨ùO¥ì¥ì
; L228
LOAD NOT  M00600	// EMERGENCY ALARM
AND NOT   D001220.6	// R_1-2 ROT R SVD BUSY
AND NOT   D001220.A	// R_1-2 ROT R WARNING
AND NOT   D001220.B	// R_1-2 ROT R MODULE ERR
AND NOT   D001220.C	// R_1-2 ROT R SVD ERR
AND NOT   M02121	// T)R_1-2 ROT R JOG-
AND NOT   M02122	// T)R_1-2 ROT R JOG+
AND NOT   M02123	// T)R_1-2 ROT R SERVO ON
AND NOT   M0312C	// R_1-2 ROT R HOME->
AND NOT   M00723	// R_1-2 ROT R NOT MV
NOT
OUT       M0162C	// R_1-2 ROT R HOLD CUT
; L229
LOAD NOT  M03120	// R_1-2 ROT R IDLE POS ->
AND NOT   M03121	// R_1-2 ROT R ROT POS ->
AND NOT   M03122	// R_1-2 ROT R BACK POS ->
AND NOT   M03123	// -
AND NOT   M03124	// -
AND NOT   M03125	// -
AND NOT   M0312A	// -
AND NOT   M01625	// R_1-2 ROT R INITIAL ->
NOT
OUTP      M0162D	// R_1-2 ROT R START 1PLS
; L230
LOAD      D001220.7	// R_1-2 ROT R A¡×A¢®¡ÆaA¢´ ¢¯I¡¤a
OUTP      M0162E	// R_1-2 ROT R POS OK PLS
; L231
LOAD      M0162D	// R_1-2 ROT R START 1PLS
LOAD      M0162F	// R_1-2 ROT R MOVE HOLD
AND NOT   M0162E	// R_1-2 ROT R POS OK PLS
AND NOT   M0162C	// R_1-2 ROT R HOLD CUT
OR LOAD
OUT       M0162F	// R_1-2 ROT R MOVE HOLD
OUT       D002220.7	// R_1-2 ROT R ABS POS MV

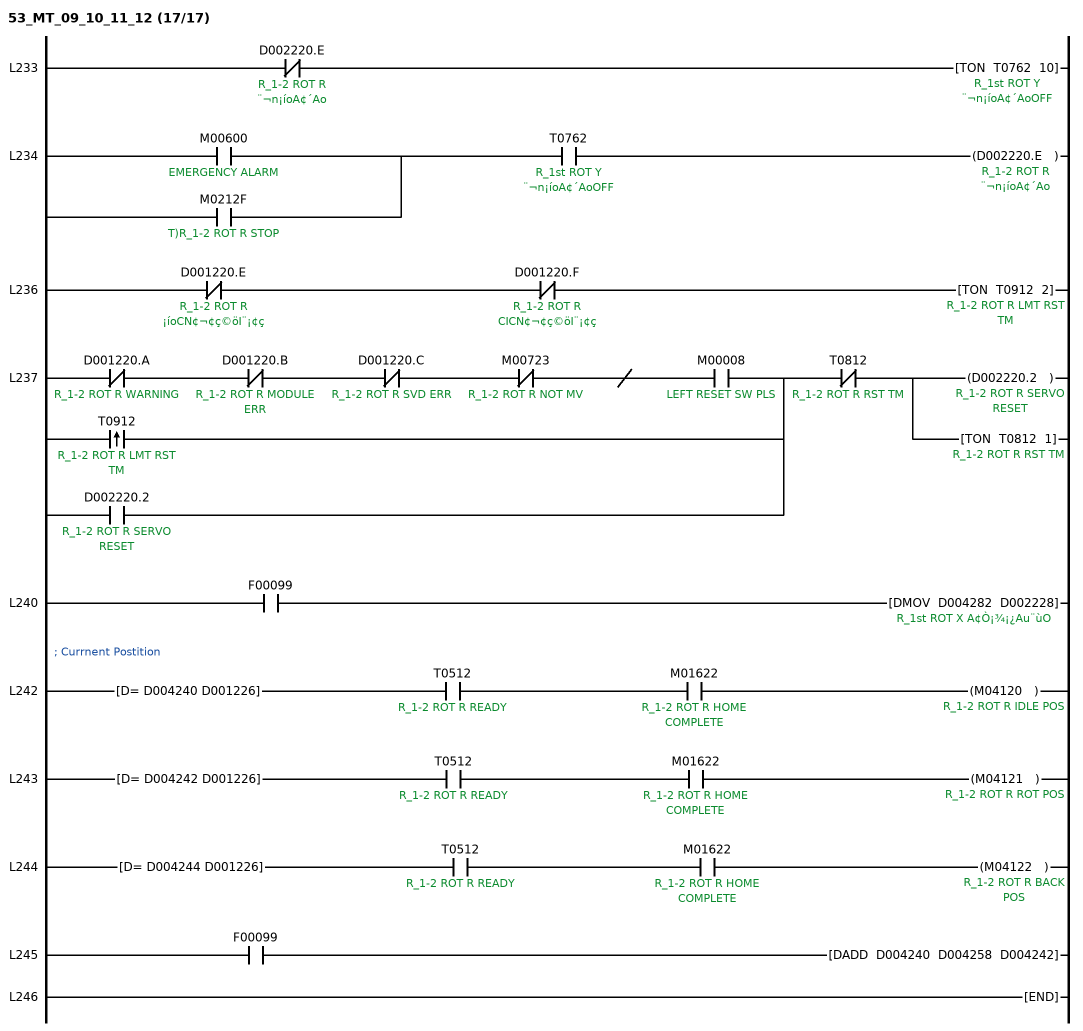
; L233
LOAD NOT  D002220.E	// R_1-2 ROT R ¨¬n¡íoA¢´Ao
TON       T0762 10	// R_1st ROT Y ¨¬n¡íoA¢´AoOFF
; L234
LOAD      M00600	// EMERGENCY ALARM
OR        M0212F	// T)R_1-2 ROT R STOP
AND       T0762	// R_1st ROT Y ¨¬n¡íoA¢´AoOFF
OUT       D002220.E	// R_1-2 ROT R ¨¬n¡íoA¢´Ao
; L236
LOAD NOT  D001220.E	// R_1-2 ROT R ¡íoCN¢¬¢ç©öI¨¡¢ç
AND NOT   D001220.F	// R_1-2 ROT R CICN¢¬¢ç©öI¨¡¢ç
TON       T0912 2	// R_1-2 ROT R LMT RST TM
; L237
LOAD NOT  D001220.A	// R_1-2 ROT R WARNING
AND NOT   D001220.B	// R_1-2 ROT R MODULE ERR
AND NOT   D001220.C	// R_1-2 ROT R SVD ERR
AND NOT   M00723	// R_1-2 ROT R NOT MV
NOT
AND       M00008	// LEFT RESET SW PLS
ORP       T0912	// R_1-2 ROT R LMT RST TM
OR        D002220.2	// R_1-2 ROT R SERVO RESET
AND NOT   T0812	// R_1-2 ROT R RST TM
OUT       D002220.2	// R_1-2 ROT R SERVO RESET
TON       T0812 1	// R_1-2 ROT R RST TM
; L240
LOAD      F00099
DMOV      D004282 D002228	// R_1st ROT X A¢Ò¡¾¡¿Au¨ùO
// Currnent Postition
; L242
LOADD=    D004240 D001226
AND       T0512	// R_1-2 ROT R READY
AND       M01622	// R_1-2 ROT R HOME COMPLETE
OUT       M04120	// R_1-2 ROT R IDLE POS
; L243
LOADD=    D004242 D001226
AND       T0512	// R_1-2 ROT R READY
AND       M01622	// R_1-2 ROT R HOME COMPLETE
OUT       M04121	// R_1-2 ROT R ROT POS
; L244
LOADD=    D004244 D001226
AND       T0512	// R_1-2 ROT R READY
AND       M01622	// R_1-2 ROT R HOME COMPLETE
OUT       M04122	// R_1-2 ROT R BACK POS
; L245
LOAD      F00099
DADD      D004240 D004258 D004242
; L246
END

PROGRAM 54_MT_13_14_15_16 (task: ¨ö¨¬A¥ì CA¡¤I¡¾¡¿¡¤¡Í)

